VAR_INPUT
	ParamTempoTimeout				: TIME := T#20S;		(* (s) Tempo before timeout. *)
	IN_Directory 					: T_maxstring := 'C:\TwinCAT\Functions\Annex_Fonctions\SendEmail\';	// Directory of the SMTP.Exe file. 
	IN_Reset_OPC					: BOOL;					// Reset Mail server and alarms. 
	IN_Restart_Service_OPC			: BOOL;					// Restart SMTP services. 
	IN_ChangePhoneMailInfos_OPC		: BOOL;					// Change users Info (mails, name, Lvl, ... ) 
	FIFO							: FB_DBDatasetFifo;		// Buffer of the alarmes). 
	
END_VAR

VAR_OUTPUT
	OUT_Completed					: BOOL;		// Juste un trig pour dire que c'est fini. Written by the SMTP.Exe
	OUT_Error						: BOOL;		// Tant qu'il y a une erreur. Written by the SMTP.exe
	OUT_Busy						: BOOL;		// Envoi en cours. 
	OUT_NbMailSent 					: UINT;	// Number of mail being sent. 
END_VAR

VAR PERSISTENT
	AX_MailAddr						: ARRAY[1..CstNbUser] OF STRING(255);	//Contient tous les numéros des utilisateurs
	AX_Subscribed					: ARRAY[1..CstNbUser] OF BOOL		;	// List of subscription. 
	AX_NomUtili						: ARRAY[1..CstNbUser] OF STRING(50)	;	// List of user names. 
	AX_User_LVL						: ARRAY[1..CstNbUser] OF WORD;			//Contient tous les niveau d'adhésion des utilisateurs.
END_VAR

VAR_INPUT PERSISTENT
	ParamTempoRetry					: TIME := T#1M;  (* (s) Tempo before send email retry *) 
	ParamNetID						: STRING :='' ; (* AMS Net ID where the SMTP.exe file is stored *)
END_VAR

VAR

	// M_AlarmManager 
	MesDataExd.MesData			: ServerMail;
	RS_AlarmDestinator		: RS;
	
	// M_Write Param	
	bAlarmNoDestinator		: BOOL;
	bSendMail				: BOOL;
	
	bWriteParam				: BOOL;
	Body					: T_MaxString;
	MailAddr				: T_MaxString;
	MesTimeStamp			: STRING(17);	
	CalTimeStamp			: STRING(255);

	//M_Send
	SendMail				: NT_StartProcess;
	
	//M_OPC
	Trig_OPC				: R_TRIG;
	RS_OPC					: RS;
	Trig_Reset				: R_TRIG;

	KK						: UINT;
	NbDest					: INT;
	TON_Retry				: TON;
	Old_Count				: UDINT;
	R_TRIG_Retry			: R_TRIG;
	
END_VAR

M_AlarmManager();
M_OPC();
M_Evaluate();

IF IN_Reset_OPC THEN
	M_Reset();
END_IF
TON_Retry(IN := Old_Count = fifo.nCount AND NOT R_TRIG_Retry.Q, pt := ParamTempoRetry);

R_TRIG_Retry(clk := TON_Retry.Q);
IF old_count <> fifo.nCount THEN
	Old_Count := fifo.nCount;
END_IF
bWriteParam := fifo.nCount > 0; 	// if the buffer is not empty, send mail. 
fifo.A_Get();	// Get the next alarm to send. 

MesTimeStamp := CONCAT(REPLACE(STR1:= left(str := FIFO.Out.TimeStamp_Act, 16), STR2 := ' ', L := 1, P := 11), ' ') ;
ReplaceAll( In_StringTosearch := MesTimeStamp, In_StringToFind := '/', IN_StringToReplace := '-', OUT_StringToSearch => CalTimeStamp);

Body := concat(left(FIFO.Out.Message, 125),SEL(FIFO.Out.Value, ' : Desactive"',' : Active"')) ; 
Body := concat( STR1:= UINT_TO_STRING(FIFO.Out.ID) , STR2:= concat(STR1:=' ,' , STR2:=Body )) ; 
Body := concat( STR1:= 'ID:' , STR2:=Body ) ; 
Body := concat('"', Concat(CalTimeStamp,Body));


MailAddr := '"';
NbDest := 0;
FOR KK := 1 TO CstNbUser DO
	IF AX_Subscribed[KK] AND AX_MailAddr[KK] <> '' AND (AX_User_LVL[KK] AND Fifo.out.Alarms_LVL)>0 THEN		// If user is subscribed to this alarm, add his mail adress to the list. 
		IF MailAddr = '"' THEN
			MailAddr := concat('"', AX_MailAddr[KK]);	// Initialize first sender. 
		END_IF
		NbDest := NbDest + 1;
	END_IF
END_FOR

IF NbDest >0 THEN
	IF NbDest>1 THEN
		FOR KK := 1 TO CstNbUser DO
			IF AX_Subscribed[KK] AND MailAddr <> AX_MailAddr[KK] AND (AX_User_LVL[KK] AND Fifo.out.Alarms_LVL)>0 THEN
				MailAddr := concat(concat(MailAddr, ', '), AX_MailAddr[KK]);		// append other mail adress if several users subsribed to this alarm. 
			END_IF
		END_FOR
	END_IF
	MailAddr := concat(MailAddr, '" ');
	bSendMail := TRUE;
	bAlarmNoDestinator	:= FALSE;
ELSE 
	bAlarmNoDestinator	:= TRUE;
	bSendMail 			:= FALSE;

END_IF	

SendMail
(
	NETID := ParamNetID,
	PATHSTR := concat(IN_Directory, 'SMTP.exe'),
	DIRNAME := IN_Directory,
	COMNDLINE := concat(str1 := MailAddr, str2 := body),
	start := bSendMail AND bWriteParam and not TON_Retry.Q
);

IF OUT_Completed THEN 
	SendMail(start := FALSE);
	OUT_Completed := FALSE;
	OUT_NbMailSent := OUT_NbMailSent + 1;

	bSendMail := FALSE;
	FIFO.A_Remove();
END_IF	

IF OUT_NbMailSent > 30000 THEN
	OUT_NbMailSent := 0;
END_IF

METHOD M_AlarmManager
VAR
	
	FB_AlarmCodeManager : FB_AlarmCodeManager;

END_VAR
// Gestion des alarmes internes au code

RS_AlarmDestinator(SET:= bAlarmNoDestinator , RESET1:= IN_Reset_OPC ) ; 

FB_AlarmCodeManager
(
	bAlarm1 := RS_AlarmDestinator.Q1,			// No recipient for at least one alarm
	bAlarm2 := OUT_Error,						// Out Error to send mail
	bAlarm3 := SendMail.ERR,					// Execution of SenMail.exe did not work. 
	bAlarm4 := FIFO.bOverwrite,					// Fifo Overflow
	bAlarm5 :=FALSE,							//
	bAlarm6 :=FALSE,    						//
	bAlarm7 :=FALSE,    						//
	bAlarm8 :=FALSE,    						//
	bAlarm9 :=FALSE,    						//
	bAlarm10 :=FALSE,   						//
	bAlarm11 :=FALSE,   						//
	bAlarm12 :=FALSE,   						//
	bAlarm13 :=FALSE,   						//
	bAlarm14 :=FALSE,   						//
	bAlarm15 :=FALSE,							//	
	wAlarmCode =>MesData.MesAlarmCode
);
END_METHOD

METHOD M_Evaluate
VAR 
END_VAR

Mesdata.AX_MailAddr		:= AX_MailAddr			;
Mesdata.AX_Subscribed	:= AX_Subscribed	    ;
MesData.AX_NomUtili		:= AX_NomUtili		    ;
MesData.OUT_NbMailSent	:= OUT_NbMailSent		;
MesData.AX_UserLVL		:= AX_User_LVL		    ;
END_METHOD

METHOD M_Init : BOOL
VAR_INPUT
END_VAR
END_METHOD

METHOD M_OPC : BOOL
VAR

END_VAR
Trig_OPC(CLK := IN_ChangePhoneMailInfos_OPC);
RS_OPC(SET:= Trig_OPC.Q);

//TrigRestartService(CLK := IN_Restart_Service_OPC);
//FUN_RestartStunnel(IN_Start := TrigRestartService.Q, IN_Directory := IN_Directory);


IF RS_OPC.Q1 THEN
	// Numéro de téléphone
	AX_MailAddr := OpcUa.AllValueW.AX_MailAddr_OPC;
	
	// Nom d'utilisateur
	AX_NomUtili	:= OpcUa.AllValueW.AX_NamesUsers_OPC;
	
	// User LVL . 
	AX_User_LVL := OpcUa.AllValueW.AX_UserLVL;
	
	// Mise a jour de la liste des subscribed
	AX_Subscribed := OpcUa.AllValueW.AX_SubscribedMail_OPC;

	RS_OPC(RESET1:= TRUE);
	RS_OPC(Reset1 := FALSE);
END_IF

Trig_Reset(CLK := IN_Reset_OPC);
IN_Reset_OPC := Trig_Reset.Q;
END_METHOD

METHOD M_Reset : BOOL
VAR_INPUT
END_VAR
VAR
	

END_VAR
FIFO.A_Reset();
IN_Reset_OPC 			:= FALSE;
bAlarmNoDestinator 		:= FALSE ;	
bSendMail				:= FALSE;
SendMail(Start:= FALSE ) ;
END_METHOD

END_PROGRAM

// ---- 00_FunctionsBlocks/Communication/ModbusRTU/CheckStruct.TcPOU
FUNCTION CheckStruct : BOOL
//Allows to compare 2 Struct_InputRTU, TRUE if struct are the same
VAR_INPUT
	InStruct1 : Struct_InputRTU;
	InStruct2 : Struct_InputRTU;
END_VAR
VAR
	bCompareBuffer 	: BOOL := TRUE;
	KK 				: UINT;
	AdrNull			: Pointer to array[1..125] of word;
END_VAR

IF InStruct1.InBuffer <> adrNull AND instruct2.InBuffer <> AdrNull THEN
	CheckStruct:= MEMCMP(pBuf1 := ADR(instruct1), pBuf2 := ADR(InStruct2), n := SIZEOF(InStruct1)) = 0;

	//FOR KK := 1 TO 125 DO
	//	bCompareBuffer := bCompareBuffer AND (InStruct1.InBuffer^[KK] = InStruct2.InBuffer^[KK]);
	//END_FOR
	//
	//
	//CheckStruct :=(InStruct1.InStartAddr	= InStruct2.InStartAddr	AND InStruct1.InQuantity	= InStruct2.InQuantity	AND InStruct1.InUnitID	    = InStruct2.InUnitID	AND  bCompareBuffer AND InStruct1.InFunction	= InStruct2.InFunction	);
END_IF

END_FUNCTION

// ---- 00_FunctionsBlocks/Communication/ModbusRTU/FB_ModbusRTU.TcPOU
FUNCTION_BLOCK FB_ModbusRTU
// Send Modbus Read Request for the first element of the buffer . Then remove the first line when executed ( busy)  and move all the other line to the left. Position 2 becomes position 1 , ...
VAR CONSTANT
	NbElementsBuffer				: UINT := 20;
	
END_VAR

VAR
	Buffer 							: ARRAY[1..NbElementsBuffer] OF Struct_InputRTU ; // Buffer to store actions
	Priority 						: ARRAY[1..NbElementsBuffer] OF UINT; // Array to store priorities
	InitialStruct 					: Struct_InputRTU;
	bInit 							: BOOL;
	ReadRTU1						: FB_ReadModbusRTU_V2;

	KK : UINT;
	
	pBoolNull						: BOOL;
	pIntNull						: INT;
	pArrayNull						: BYTE;

	R_TRIG_Error					: R_TRIG ;
	
END_VAR

IF NOT bInit THEN
	// Empty all structures . 
	M_Init();
ELSE
	
		// ATTENTION , IL NE FAUT PAS ENVOYER UN NOUVEAU MODBUS TANT QUE LE PRECEDENT N EST PAS FINI DE TRAITER .DE MEME IL NE FAUT PAS QUE LE CYCLE D AJOUT DU FIFO SOIT PLUS RAPIDE QUE LE TRAITEMENT DU RTU 
		// TEmpo de 30 s apres une alarmes avant de refaire un essai . il ne faudrait pas que ca bloque les autres commandes .  

		IF priority[1] <> 0 THEN

			ReadRTU1(
				InClockRead := TRUE,
				InStartAddr := Buffer[1].InStartAddr,
				InQuantity := Buffer[1].InQuantity,
				InUnitID := Buffer[1].InUnitID,
				InTimeout := T#500MS,
				InAddrDest := Buffer[1].InBuffer,
				InFunctionRead := Buffer[1].InFunction
			);
		END_IF
		
		
		
		MEMCPY(destAddr := Buffer[1].OutBusy, srcAddr := ADR(ReadRTU1.OutBusy), n := SIZEOF(ReadRTU1.OutBusy));		

		//R_TRIG_Error(CLK:= ReadRTU1.OutErrorMbRead) ; 
		
		IF ReadRTU1.OutbCompleted OR ReadRTU1.OutErrorMbRead THEN	// La lecture s 'est terminée par une erreur ou correcteemnt, on passe à l'element du buffer suivant . 
			MEMCPY(destAddr := Buffer[1].OutError, srcAddr := ADR(ReadRTU1.OutErrorMbRead), n := SIZEOF(ReadRTU1.OutErrorMbRead)); // Copy the errOR  
			MEMCPY(destAddr := Buffer[1].OutErrorId, srcAddr := ADR(ReadRTU1.OutErrorId), n := SIZEOF(ReadRTU1.OutErrorId));
			MEMCPY(destAddr := Buffer[1].OutCompleted, srcAddr := ADR(ReadRTU1.OutbCompleted), n := SIZEOF(ReadRTU1.OutbCompleted));	
			ReadRTU1.InClockRead := FALSE ; 
			ReadRTU1.Reset		:= TRUE ; 
			M_DeleteAction(InLigne := 1);
			//R_TRIG_Error(CLK:= FALSE ) ; 
			
		END_IF
END_IF

METHOD M_AddAction_FIFO : UINT //Method to add an element with a priority using FIFO strategy

VAR_INPUT
	InStruct 		: Struct_InputRTU;		// Structure input
	InPriority 		: UINT;					// Strategy input
END_VAR
VAR_OUTPUT
	OutBusy 		: BOOL;					// Output state of the Method
	OutError 		: BOOL;					// Output error of the Method
	OutErrorID 		: UINT;					//1: Empty input 2: Full Buffer
	OutCompleted 	: BOOL;					// Output state of the Method : not busy and no error
END_VAR
VAR
	KK 				: UINT;
	LineToDelete	: UINT;
END_VAR
OutError 	:= FALSE;
OutBusy 	:= TRUE;

IF NOT (CheckStruct(InStruct1 := InitialStruct, InStruct2 := InStruct)) AND InPriority <> 0 THEN 			// Check that we don't input an empty value
	IF CheckStruct(InStruct1 := buffer[NbElementsBuffer], InStruct2 := InitialStruct) THEN 			// Check that the buffer isn't already full
		FOR KK := 1 TO NbElementsBuffer - 1 DO
			IF NOT CheckStruct(InStruct1 := buffer[NbElementsBuffer-KK], InStruct2 := InitialStruct) AND Priority[NbElementsBuffer-KK] > InPriority THEN 			// If the next position isn't empty  
				buffer[NbElementsBuffer-KK+1] := buffer[NbElementsBuffer-KK]; 		// I replace this position by the next  ( CE PREMIER IF N EST PAS EXECUTER SI TOUTES LES PRIORITES SONT IDENTIQUES . )
				Priority[NbElementsBuffer -KK +1 ] := Priority[NbElementsBuffer-KK];
			ELSE
				IF NOT CheckStruct(InStruct1 := buffer[NbElementsBuffer-KK], InStruct2 := InitialStruct) THEN		// Detect for buffer element that is not empty and assign new element to read to it. 
					buffer[NbElementsBuffer-KK+1] 	:= InStruct;
					M_AddAction_FIFO 				:= NbElementsBuffer-KK+1;
					Priority[NbElementsBuffer-KK+1] := InPriority;
					OutCompleted 		:= TRUE;
					EXIT ;
				END_IF
			END_IF
		END_FOR
		IF NOT Outcompleted THEN
			buffer[1] := InStruct;
			Priority[1] := InPriority;
			OutCompleted := TRUE;
			M_AddAction_Fifo := 1;
		END_IF
	ELSE
		OutErrorID 	:= 2;
		OutError 	:= TRUE;
	END_IF
ELSE
	OutErrorID 	:= 1;
	OutError 	:= TRUE;
END_IF
IF M_VerifActions(OutLigne=>LineToDelete) THEN	// Verifie si il  n ya pas deux fois la meme ligne , sinon, supprime les lignes en doubles . En pratique, forcement la derniere ligne . 
	M_DeleteAction(InLigne := LineToDelete);
END_IF
OutBusy := FALSE;
END_METHOD

METHOD M_DeleteAction : BOOL
VAR_INPUT
	InLigne 	: UINT;			// Input Ligne to delete
END_VAR
VAR_OUTPUT
	OutBusy 		: BOOL;					// Output state of the Method
	OutError 		: BOOL;					// Output error of the Method
	OutErrorID 		: UINT;					// 1: InLigne greater than Buffer size, 2: The buffer ligne is already empty, 3: The buffer is full
	OutCompleted 	: BOOL;					// Output state of the Method : not busy and no error
	
END_VAR

VAR
	KK 				: UINT;
END_VAR
IF InLigne <= NbElementsBuffer THEN // Check the InLigne is in the range of the buffer
	IF NOT checkstruct(InStruct1 := buffer[InLigne], InStruct2 := InitialStruct) THEN	// Check that the buffer ligne is not already empty
		IF checkstruct(InStruct1 := buffer[NbElementsBuffer], InStruct2 := InitialStruct)THEN //check that the buffer is not full
			FOR KK := InLigne TO NbElementsBuffer -1 DO
				Buffer[KK] := buffer[KK + 1] ;
				Priority[KK] := Priority[KK + 1] ;
			END_FOR
		ELSE
			OutError := TRUE;
			OutBusy := FALSE;
			OutCompleted := FALSE;
			OutErrorID := 3;
		END_IF
	ELSE
		OutError := TRUE;
		OutCompleted := FALSE;
		OutBusy := TRUE;
		OutErrorID := 2;
		
	END_IF
ELSE
	OutCompleted := FALSE;
	OutError := TRUE;
	OutBusy := FALSE;
	OutErrorID := 1;
END_IF
END_METHOD

METHOD M_Init : BOOL
VAR
	InStruct : Struct_InputRTU;
END_VAR

// Initialize the structure with empty elements. 

InitialStruct.InBuffer := ADR(pArrayNull);
InitialStruct.OutBusy := ADR(pBoolNull);
InitialStruct.OutCompleted := ADR(pBoolNull);
InitialStruct.OutError := ADR(pBoolNull);
InitialStruct.OutErrorId := ADR(pIntNull);
FOR KK := 1 TO NbElementsBuffer DO 
	Buffer[KK] := InitialStruct;
END_FOR	

bInit := TRUE;
END_METHOD

METHOD M_VerifActions : BOOL // Verifies there is not repeat in the liste : TRUE = At least 2 elements are the same
VAR_OUTPUT
	OutLigne 	 : UINT;
END_VAR

VAR
	KK: UINT;
	JJ: UINT;
	CheckStructValue : BOOL;
END_VAR
FOR KK := 1 TO NbElementsBuffer DO
	FOR JJ := 1 + KK TO NbElementsBuffer DO
		IF CheckStruct(InStruct1 := InitialStruct, instruct2 := buffer[KK]) THEN
			EXIT;
		ELSE
			CheckStructValue :=  checkstruct(InStruct1 := buffer[JJ], InStruct2 := buffer[KK]);
			M_VerifActions := M_VerifActions OR (CheckStructValue ) ;
			OutLigne := SEL(CheckStructValue AND Priority[KK]> priority[JJ], KK, JJ);
		END_IF
	END_FOR
END_FOR
END_METHOD

END_FUNCTION_BLOCK

// ---- 00_FunctionsBlocks/Communication/ModbusRTU/FB_ReadModbusRTU_V2.TcPOU
FUNCTION_BLOCK FB_ReadModbusRTU_V2
/////////////////////////////////////////////////////////////////////// 
///////Read Modbus RTU on Rising Edge of Trigger ClockRead ////////
//If there is lost of communication, ParamNbAlms then if still 
//error wait ParamTimeRetry then loop 
//Version : V1.1
///////////////////////////////////////////////////////////////////////

VAR_INPUT
	InClockRead 			: BOOL;  		// Boolean to start the read
	InStartAddr				: WORD;  		// First address of the block
	InQuantity			    : WORD;	 		// Quantity of registers to read
	InUnitID				: BYTE ; 		// Unit Id of the Slave to be read
	InTimeout 				: TIME:=T#2S;   // Timeout param for the read
	InAddrDest		        : POINTER TO BYTE;
	InFunctionRead          : UINT;          // 0 := ReadInputRegs, 1 := ReadRegs 
	ParamEnableRetryPause	: BOOL ; 
	Reset					: BOOL ;
END_VAR

VAR_OUTPUT
	OutErrorMbRead  		: BOOL; 	                // Alarm if three modbus attempts failed.
	OutBusy					: BOOL;					    //Busy
	OutErrorId				: INT;            //Id number of the error based on TC
	OutbCompleted			: BOOL;
	TmpError				: BOOL;	
END_VAR

VAR
	//Parameters
	ParamNbAlms				: UINT := 3;				// Parameter for the number of retries before the alarme
	ParamTimeRetry 			: TIME:=T#30S;				//Time to wait before a retry
	
	//Instantiation of FB
	MB 						: ModbusRtuMaster_PcCOM; 		// Multiple registers reading FROM SUB9 Interface
	MB_EL					: ModbusRtuMasterV2_KL6x22B;  // Multiple registers reading FROM EL6021 Interface
	R_TRIG          		: R_TRIG; 					// Rising edge detection for the trigger.
	TempoRetry      		: TP;
	
	//Variables of the code 
	Step            		: INT; 		    			// Grafcet step
	AlarmCounter    		: UINT; 					// Alarm Counter. Incremennted if modbus errOR  Alarm if counter =3 , resetable.  
	bRetry          		: BOOL:= FALSE; 			// Boolean to denote the retries
	
	TmpBusy					: BOOL;
	TmpErrorId				: INT;	
	
	TON_ReadRTU						: TON; 
END_VAR

OutbCompleted:= FALSE;
// RESET //
	IF Reset THEN 
			AlarmCounter		:= MAX(0,AlarmCounter-1) ;	// on enleve 1 au compteur pour supprimer l'alamrme. 
			OutErrorId 			:= 0 ; 
			OutErrorMbRead 	:=FALSE;
			Reset 				:= FALSE;
	END_IF
	
// ALARM MANAGEMENT //
TempoRetry(PT := ParamTimeRetry);
IF AlarmCounter = ParamNbAlms THEN 
	OutErrorMbRead 	:=TRUE;
	bRetry := SEL(ParamEnableRetryPause , FALSE ,  TRUE);		// False = disable retry 	
ELSE
	bRetry := FALSE;
	
END_IF

	// MODBUS SEQUENCE //
	CASE step OF
		0://Idle
			R_TRIG(CLK := InClockRead);
			IF R_TRIG.Q THEN 
				R_TRIG(CLK := FALSE);
				Step :=1;
				OutBusy         := TRUE;
			END_IF
		1 ://Processing Reply  
			TON_ReadRTU(IN:= TRUE , PT:= InTimeout + T#100MS ) ; // Overlay timeout . 
	    	CASE InFunctionRead OF
				1: 
					MB_EL.ReadCoils
					(
						UnitID := InUnitId, 
						Quantity := InQuantity, 
						MBAddr := InStartAddr, 
						cbLength := 2* InQuantity, 
						pMemoryAddr := InAddrDest, 
						Execute := TRUE, 
						Timeout := InTimeout,
						Error => TmpError,
						Busy => TmpBusy,
						ErrorId => TmpErrorId,
					);	
				2:
					MB_EL.ReadInputStatus
					(
						UnitID := InUnitId, 
						Quantity := InQuantity, 
						MBAddr := InStartAddr, 
						cbLength := 2* InQuantity, 
						pMemoryAddr := InAddrDest, 
						Execute := TRUE, 
						Timeout := InTimeout,
						Error => TmpError,
						Busy => TmpBusy,
						ErrorId => TmpErrorId,
					);	
				3:
					MB_EL.ReadRegs
					(
						UnitID := InUnitId, 
						Quantity := InQuantity, 
						MBAddr := InStartAddr, 
						cbLength := 2* InQuantity, 
						pMemoryAddr := InAddrDest, 
						Execute := TRUE, 
						Timeout := InTimeout,
						Error => TmpError,
						Busy => TmpBusy,
						ErrorId => TmpErrorId,
					  );
				4:
					MB_EL.ReadInputRegs
					(
						UnitID := InUnitId, 
						Quantity := InQuantity, 
						MBAddr := InStartAddr, 
						cbLength := 2* InQuantity, 
						pMemoryAddr := InAddrDest, 
						Execute := TRUE, 
						Timeout := InTimeout,
						Error => TmpError,
						Busy => TmpBusy,
						ErrorId => TmpErrorId,
					);
				5:
					MB_EL.WriteSingleCoil
					(
						UnitID := InUnitId, 
						Quantity := InQuantity, 
						MBAddr := InStartAddr, 
						cbLength := 2* InQuantity, 
						pMemoryAddr := InAddrDest, 
						Execute := TRUE, 
						Timeout := InTimeout,
						Error => TmpError,
						Busy => TmpBusy,
						ErrorId => TmpErrorId,
					);
				6:
					MB_EL.WriteSingleRegister
					(
						UnitID := InUnitId, 
						Quantity := InQuantity, 
						MBAddr := InStartAddr, 
						cbLength := 2* InQuantity, 
						pMemoryAddr := InAddrDest, 
						Execute := TRUE, 
						Timeout := InTimeout,
						Error => TmpError,
						Busy => TmpBusy,
						ErrorId => TmpErrorId,
					);
				15:
					MB_EL.WriteMultipleCoils
					(
						UnitID := InUnitId, 
						Quantity := InQuantity, 
						MBAddr := InStartAddr, 
						cbLength := 2* InQuantity, 
						pMemoryAddr := InAddrDest, 
						Execute := TRUE, 
						Timeout := InTimeout,
						Error => TmpError,
						Busy => TmpBusy,
						ErrorId => TmpErrorId,
					);
				16:
					MB_EL.WriteRegs
					(
						UnitID := InUnitId, 
						Quantity := InQuantity, 
						MBAddr := InStartAddr, 
						cbLength := 2* InQuantity, 
						pMemoryAddr := InAddrDest, 
						Execute := TRUE, 
						Timeout := InTimeout,
						Error => TmpError,
						Busy => TmpBusy,
						ErrorId => TmpErrorId,
					);
			END_CASE
			
			IF NOT (TmpBusy) AND NOT (TmpError) THEN
				TempoRetry(In:= FALSE);
				TON_ReadRTU(IN:= FALSE ) ; 
				MB_EL.ReadInputRegs(Execute:= FALSE);
				MB_EL.ReadRegs(Execute:= FALSE);
				MB_EL.ReadCoils(Execute:= FALSE);
				MB_EL.ReadInputStatus(Execute:= FALSE);
				MB_EL.WriteSingleCoil(Execute:= FALSE);
				MB_EL.WriteSingleRegister(Execute:= FALSE);
				MB_EL.WriteMultipleCoils(Execute:= FALSE);
				MB_EL.WriteRegs(Execute:= FALSE);
				OutErrorId 		:= 0;
				OutErrorMbRead	:= FALSE;
				AlarmCounter	:= 0; // Reset counter after successful modbus read. 
				OutbCompleted 	:= TRUE ; 
				Step 			:= 0;
				OutBusy         := FALSE;
			ELSIF ((NOT (TmpBusy) AND TmpError) OR TON_ReadRTU.Q)  AND NOT(bRetry) THEN

				TempoRetry(In:= FALSE);
				bRetry := FALSE;
				MB_EL.ReadCoils(Execute:= FALSE);
				MB_EL.ReadInputRegs(Execute:= FALSE);
				MB_EL.ReadInputStatus(Execute:= FALSE);
				MB_EL.ReadRegs(Execute:= FALSE);
				MB_EL.WriteSingleCoil(Execute:= FALSE);
				MB_EL.WriteSingleRegister(Execute:= FALSE);
				MB_EL.WriteMultipleCoils(Execute:= FALSE);
				MB_EL.WriteRegs(Execute:= FALSE);
				AlarmCounter 	:= MIN(AlarmCounter + 1,3) ; 
				OutErrorId		:= SEL(TON_ReadRTU.Q , TmpErrorId ,250 );
				Step 			:= 0;
				TON_ReadRTU(IN:= FALSE ) ; 
				OutBusy         := FALSE;
			ELSIF NOT (TmpBusy) AND TmpError AND bRetry THEN
				MB_EL.ReadInputRegs(Execute:= FALSE);
				MB_EL.ReadRegs(Execute:= FALSE);
				MB_EL.ReadCoils(Execute:= FALSE);
				MB_EL.ReadInputStatus(Execute:= FALSE);
				MB_EL.WriteSingleCoil(Execute:= FALSE);
				MB_EL.WriteSingleRegister(Execute:= FALSE);
				MB_EL.WriteMultipleCoils(Execute:= FALSE);
				MB_EL.WriteRegs(Execute:= FALSE);
				step := 2;
				OutBusy         := FALSE;
			END_IF	
		2: 
			TempoRetry(In:= TRUE);		// LEAVE SOME TIME BEFORE NEW ATTEMPT . 
			IF NOT(TempoRetry.Q) THEN
				TempoRetry(In:= FALSE);
				//AlarmCounter := 0;
				step := 0;
				
			END_IF
			
	END_CASE

END_FUNCTION_BLOCK

// ---- 00_FunctionsBlocks/Communication/ModbusRTU/Sample_ModbusRTU.TcPOU
PROGRAM Sample_ModbusRTU
VAR
	ModbusRTU				: FB_ModbusRTU;
	MesBlock				: ARRAY[1..8] OF ARRAY[1..120] OF WORD;	
	AX_Addr					: ARRAY[1..8] OF UINT 	:= [1,		1,		1,		1,		1, 		1, 		1, 		1];
	AX_Qty					: ARRAY[1..8] OF UINT	:= [1,		1,		1,		1,		1, 		1, 		1, 		1];
	AX_UnitId				: ARRAY[1..8] OF BYTE	:= [1,		1,		1,		1,		1, 		1, 		1, 		1];
	AX_Function				: ARRAY[1..8] OF UINT	:= [1,		2,		3,		4,		5, 	 	6, 	 	15, 	16];	
	AX_Priority				: ARRAY[1..8] OF UINT	:= [1,		1,		1,		1,		1, 	 	1, 	 	1, 		1 ];
	AX_bStart				: ARRAY[1..8] OF BOOL;
	MbStruct				: ARRAY[1..8] OF Struct_InputRTU;	
	
	KK: INT;
END_VAR

ModbusRTU();

FOR KK := 1 TO 8 DO 
	MbStruct[KK].InBuffer := ADR(MesBlock[KK]);
	MbStruct[KK].InFunction := AX_Function[KK];
	MbStruct[KK].InQuantity := AX_Qty[KK];
	MbStruct[KK].InStartAddr := AX_Addr[KK];
	MbStruct[KK].InUnitID := AX_UnitId[KK];
END_FOR


IF CalLocalTimeStruct.wSecond MOD 5 = 0 THEN
	FOR KK := 1 TO 8 DO
		IF AX_bStart[KK] THEN
			ModbusRTU.M_AddAction_FIFO(InStruct := MbStruct[KK], InPriority := AX_Priority[KK]);
		END_IF
	END_FOR
	
END_IF

END_PROGRAM

// ---- 00_FunctionsBlocks/Communication/ModbusTCP/FB_ModbusRead.TcPOU
FUNCTION_BLOCK FB_ModbusRead
////////////////// 
// Read Modbus TCP/IP on Rising Edge of Trigger ClockRead. Returns alarm and stop modbus Read after three consecutive Modbus attempts that failed. 
//////////////////

VAR_INPUT
	
	// Modbus ReadRegs FB inputs
	pDestAddr 	: POINTER TO BYTE ; // Pointer to variable in which the read data have to be stored
	sIPAddr 	: STRING(15);		// Modbus server device IP adress
	tTimeout 	: TIME;				// Timeout
	nTcpPort 	: UINT;
	nQuantity 	: WORD;				// Quantity of words to be read
	nMBAddr 	: WORD ;			// Starting Register adress
	
	cbLength 	: UDINT;			// Length of variable to host the read data
	nUnitID 	: BYTE;				// Unit ID in case of serial connexion after modbus server. Usually equals to 1
	
	ClockRead	: BOOL; 			// Rising Edge Modbus Trigger
	Reset		: BOOL; 			// Reset Trigger to clean alarm and counter.
	
	ParamTimeRetry 			: TIME:=T#30S;				//Time to wait before a retry
	ParamNbAlms				: INT := 3;				// Parameter for the number of retries before the alarme
	ParamEnableRetryPause	: BOOL ; 
	
	
END_VAR

VAR_OUTPUT
	ErrorId			: UDINT;	// Error Id returned by FB ( see ADS error Code ) . 
	
	Busy			: BOOL ;	// FB busy to proceed command
	ModbusReadAlarm	: BOOL; 	// Alarm if three modbus attempt failed.
	OUT_NbRead		: UDINT;
END_VAR

VAR
	R_TRIG 				: R_TRIG; 			// Rising edge detection for the trigger.
	FB_MBReadRegs 		: FB_MBReadRegs; 	// Multiple registers reading
	
	Step				: INT; 				// Grafcet step
	AlarmCounter		: INT; 				// Alarm Counter. Incremennted if modbus errOR  Alarm if counter =3 , resetable.  

	TempoRetry      		: TP;

	bRetry          		: BOOL:= FALSE; 			// Boolean to denote the retries	
END_VAR

// ALARM MANAGEMENT //
TempoRetry(PT := ParamTimeRetry);
	IF AlarmCounter=ParamNbAlms THEN 
		ModbusReadAlarm 	:=TRUE;
		bRetry := SEL(ParamEnableRetryPause , FALSE ,  TRUE);		// False = disable retry 		
	ELSE
		ModbusReadAlarm := FALSE;
		ErrorId			:= 0;
		bRetry := FALSE;		// False = disable retry 	
	END_IF


// MODBUS SEQUENCE //
CASE Step OF 
	0:
		R_TRIG(CLK :=ClockRead);
		
		IF R_TRIG.Q THEN 
			Step :=1;
			Busy := TRUE;
			OUT_NbRead := 0;
		END_IF
	1:
	   FB_MBReadRegs(
	  			sIPAddr:= sIPAddr , 
				nTCPPort:= nTcpPort ,
				nUnitID:= nUnitID,
				nQuantity:= nQuantity,
				nMBAddr:= nMBAddr, 
				cbLength:= cbLength, 
				pDestAddr:= pDestAddr, 
				bExecute:= TRUE,
				tTimeout:= tTimeout,
				cbRead => OUT_NbRead
				);
				
		IF NOT FB_MBReadRegs.bBusy AND NOT FB_MBReadRegs.bError THEN
			FB_MBReadRegs(bExecute:= FALSE);
			AlarmCounter	:=0; // Reset counter after successful modbus read. 
			Step 			:=0;
			Busy := FALSE;
		ELSIF NOT FB_MBReadRegs.bBusy AND FB_MBReadRegs.bError AND NOT(bRetry) THEN
			FB_MBReadRegs(bExecute:= FALSE);
			AlarmCounter 	:= MIN(AlarmCounter+1,ParamNbAlms) ; 
			ErrorId			 :=FB_MBReadRegs.nErrId;
			Step 			:=0;
			Busy := FALSE;
			TempoRetry(In:= FALSE);
			bRetry := FALSE;
		ELSIF NOT FB_MBReadRegs.bBusy AND FB_MBReadRegs.bError AND bRetry THEN
			FB_MBReadRegs(bExecute:= FALSE);
			step := 2;
			Busy := FALSE;		
		END_IF	
	2: 
		TempoRetry(In:= TRUE);		// LEAVE SOME TIME BEFORE NEW ATTEMPT . 
		IF NOT(TempoRetry.Q) THEN
			TempoRetry(In:= FALSE);
			//AlarmCounter := 0;
			step := 0;
			
		END_IF
		
END_CASE

// RESET //
	IF Reset THEN 
			AlarmCounter 		:= 0 ; 
			ErrorId 			:= 0 ; 
			ModbusReadAlarm 	:=FALSE;
			Reset 				:= FALSE;
	END_IF

// BUSY //

END_FUNCTION_BLOCK

// ---- 00_FunctionsBlocks/Communication/ModbusTCP/FB_ModbusReadCoils.TcPOU
FUNCTION_BLOCK FB_ModbusReadCoils
////////////////// 
// Read Modbus TCP/IP on Rising Edge of Trigger ClockRead. Returns alarm and stop modbus Read after three consecutive Modbus attempts that failed. 
//////////////////

VAR_INPUT
	
	// Modbus ReadRegs FB inputs
	pDestAddr 	: POINTER TO BYTE ; // Pointer to variable in which the read data have to be stored
	sIPAddr 	: STRING(15);		// Modbus server device IP adress
	tTimeout 	: TIME;				// Timeout
	nTcpPort 	: UINT;
	nQuantity 	: WORD;				// Quantity of words to be read
	nMBAddr 	: WORD ;			// Starting Register adress
	
	cbLength 	: UDINT;			// Length of variable to host the read data
	nUnitID 	: BYTE;				// Unit ID in case of serial connexion after modbus server. Usually equals to 1
	
	ClockRead	: BOOL; 			// Rising Edge Modbus Trigger
	Reset		: BOOL; 			// Reset Trigger to clean alarm and counter.
	
END_VAR

VAR_OUTPUT
	ErrorId			: UDINT;	// Error Id returned by FB ( see ADS error Code ) . 
	
	Busy			: BOOL ;	// FB busy to proceed command
	ModbusReadAlarm	: BOOL; 	// Alarm if three modbus attempt failed.
	OUT_NbRead		: UDINT;
END_VAR

VAR
	R_TRIG 				: R_TRIG; 			// Rising edge detection for the trigger.
	FB_MBReadCoils 		: FB_MBReadCoils; 	// Multiple registers reading
	
	Step				: INT; 				// Grafcet step
	AlarmCounter		: INT; 				// Alarm Counter. Incremennted if modbus errOR  Alarm if counter =3 , resetable.  

	
END_VAR

// ALARM MANAGEMENT //

	IF AlarmCounter=3 THEN 
		ModbusReadAlarm 	:=TRUE;
		
	ELSE
		ModbusReadAlarm := FALSE;
		ErrorId			:= 0;
		
	END_IF


// MODBUS SEQUENCE //
CASE Step OF 
	0:
		R_TRIG(CLK :=ClockRead);
		
		IF R_TRIG.Q THEN 
			Step :=1;
			Busy := TRUE;
			OUT_NbRead := 0;
		END_IF
	1:
	   FB_MBReadCoils(
	  			sIPAddr:= sIPAddr , 
				nTCPPort:= nTcpPort ,
				nUnitID:= nUnitID,
				nQuantity:= nQuantity,
				nMBAddr:= nMBAddr, 
				cbLength:= cbLength, 
				pDestAddr:= pDestAddr, 
				bExecute:= TRUE,
				tTimeout:= tTimeout,
				cbRead => OUT_NbRead
				);
				
		IF NOT FB_MBReadCoils.bBusy AND NOT FB_MBReadCoils.bError THEN
			FB_MBReadCoils(bExecute:= FALSE);
			AlarmCounter	:=0; // Reset counter after successful modbus read. 
			Step 			:=0;
			Busy := FALSE;
		ELSIF NOT FB_MBReadCoils.bBusy AND FB_MBReadCoils.bError THEN
			FB_MBReadCoils(bExecute:= FALSE);
			AlarmCounter 	:= MIN(AlarmCounter+1,3) ; 
			ErrorId			 :=FB_MBReadCoils.nErrId;
			Step 			:=0;
			Busy := FALSE;
		END_IF
		
END_CASE

// RESET //
	IF Reset THEN 
			AlarmCounter 		:= 0 ; 
			ErrorId 			:= 0 ; 
			ModbusReadAlarm 	:=FALSE;
			Reset 				:= FALSE;
			FB_MBReadCoils		(bExecute := FALSE);
	END_IF

// BUSY //

END_FUNCTION_BLOCK

// ---- 00_FunctionsBlocks/Communication/ModbusTCP/FB_ModbusReadInput.TcPOU
FUNCTION_BLOCK FB_ModbusReadInput
////////////////// 
// Read Modbus TCP/IP on Rising Edge of Trigger ClockRead. Returns alarm and stop modbus Read after three consecutive Modbus attempts that failed. 
//////////////////

VAR_INPUT
	
	// Modbus ReadRegs FB inputs
	pDestAddr 	: POINTER TO BYTE ; // Pointer to variable in which the read data have to be stored
	sIPAddr 	: STRING(15);		// Modbus server device IP adress
	tTimeout 	: TIME;				// Timeout
	nTcpPort 	: UINT;
	nQuantity 	: WORD;				// Quantity of words to be read
	nMBAddr 	: WORD ;			// Starting Register adress
	
	cbLength 	: UDINT;			// Length of variable to host the read data
	nUnitID 	: BYTE;				// Unit ID in case of serial connexion after modbus server. Usually equals to 1
	
	ClockRead	: BOOL; 			// Rising Edge Modbus Trigger
	Reset		: BOOL; 			// Reset Trigger to clean alarm and counter.
	
END_VAR

VAR_OUTPUT
	ErrorId			: UDINT;	// Error Id returned by FB ( see ADS error Code ) . 
	
	Busy			: BOOL ;	// FB busy to proceed command
	ModbusReadAlarm	: BOOL; 	// Alarm if three modbus attempt failed.
	OUT_NbRead		: UDINT;
END_VAR

VAR
	R_TRIG 				: R_TRIG; 			// Rising edge detection for the trigger.
	FB_MBReadInputs 		: FB_MBReadInputs; 	// Multiple registers reading
	
	Step				: INT; 				// Grafcet step
	AlarmCounter		: INT; 				// Alarm Counter. Incremennted if modbus errOR  Alarm if counter =3 , resetable.  

	
END_VAR

// ALARM MANAGEMENT //

	IF AlarmCounter=3 THEN 
		ModbusReadAlarm 	:=TRUE;
		
	ELSE
		ModbusReadAlarm := FALSE;
		ErrorId			:= 0;
		
	END_IF


// MODBUS SEQUENCE //
CASE Step OF 
	0:
		R_TRIG(CLK :=ClockRead);
		
		IF R_TRIG.Q THEN 
			Step :=1;
			Busy := TRUE;
			OUT_NbRead := 0;
		END_IF
	1:
	   FB_MBReadInputs(
	  			sIPAddr:= sIPAddr , 
				nTCPPort:= nTcpPort ,
				nUnitID:= nUnitID,
				nQuantity:= nQuantity,
				nMBAddr:= nMBAddr, 
				cbLength:= cbLength, 
				pDestAddr:= pDestAddr, 
				bExecute:= TRUE,
				tTimeout:= tTimeout,
				cbRead => OUT_NbRead
				);
				
		IF NOT FB_MBReadInputs.bBusy AND NOT FB_MBReadInputs.bError THEN
			FB_MBReadInputs(bExecute:= FALSE);
			AlarmCounter	:=0; // Reset counter after successful modbus read. 
			Step 			:=0;
			Busy := FALSE;
		ELSIF NOT FB_MBReadInputs.bBusy AND FB_MBReadInputs.bError THEN
			FB_MBReadInputs(bExecute:= FALSE);
			AlarmCounter 	:= MIN(AlarmCounter+1,3) ; 
			ErrorId			 :=FB_MBReadInputs.nErrId;
			Step 			:=0;
			Busy := FALSE;
		END_IF
		
END_CASE

// RESET //
	IF Reset THEN 
			AlarmCounter 		:= 0 ; 
			ErrorId 			:= 0 ; 
			ModbusReadAlarm 	:=FALSE;
			Reset 				:= FALSE;
			FB_MBReadInputs		(bExecute := FALSE);
	END_IF

// BUSY //

END_FUNCTION_BLOCK

// ---- 00_FunctionsBlocks/Communication/ModbusTCP/FB_ModbusReadInputRegs.TcPOU
FUNCTION_BLOCK FB_ModbusReadInputRegs
////////////////// 
// Read Modbus TCP/IP on Rising Edge of Trigger ClockRead. Returns alarm and stop modbus Read after three consecutive Modbus attempts that failed. 
//////////////////

VAR_INPUT
	
	// Modbus ReadRegs FB inputs
	pDestAddr 	: POINTER TO BYTE ; // Pointer to variable in which the read data have to be stored
	sIPAddr 	: STRING(15);		// Modbus server device IP adress
	tTimeout 	: TIME;				// Timeout
	
	nTCPport	: UINT:= 502;		// TCP Port
	
	nQuantity 	: WORD;				// Quantity of words to be read
	nMBAddr 	: WORD ;			// Starting Register adress
	
	cbLength 	: UDINT;			// Length of variable to host the read data
	nUnitID 	: BYTE;				// Unit ID in case of serial connexion after modbus server. Usually equals to 1
	
	ClockRead	: BOOL; 			// Rising Edge Modbus Trigger
	Reset		: BOOL; 			// Reset Trigger to clean alarm and counter.
	
	ParamTimeRetry 			: TIME:=T#30S;				//Time to wait before a retry
	ParamNbAlms				: INT := 3;				// Parameter for the number of retries before the alarme
	ParamEnableRetryPause	: BOOL ; 
	
END_VAR

VAR_OUTPUT
	ErrorId			: UDINT;	// Error Id returned by FB ( see ADS error Code ) . 
	OUT_Completed	: BOOL ; // Reading completed successfully . 
	Busy			: BOOL ;	// FB busy to proceed command
	ModbusReadAlarm	: BOOL; 	// Alarm if three modbus attempt failed.
	
END_VAR

VAR
	R_TRIG 				: R_TRIG; 			// Rising edge detection for the trigger.
	FB_MBReadInputRegs 	: FB_MBReadInputRegs; 	// Multiple registers reading
	
	Step				: INT; 				// Grafcet step
	AlarmCounter		: INT; 				// Alarm Counter. Incremennted if modbus errOR  Alarm if counter =3 , resetable.  
	TempoRetry      		: TP;

	bRetry          		: BOOL:= FALSE; 			// Boolean to denote the retries	
	
END_VAR

// ALARM MANAGEMENT //
TempoRetry(PT := ParamTimeRetry);
	IF AlarmCounter=3 THEN 
		ModbusReadAlarm 	:=TRUE;
		bRetry := SEL(ParamEnableRetryPause , FALSE ,  TRUE);		// False = disable retry 		
	ELSE
		ModbusReadAlarm := FALSE;
		ErrorId			:= 0;
		bRetry := FALSE;		// False = disable retry 
	END_IF

OUT_Completed := FALSE ; 

// MODBUS SEQUENCE //
CASE Step OF 
	0:
		R_TRIG(CLK :=ClockRead);
		IF R_TRIG.Q THEN 
			Step :=1;
			Busy := TRUE;
		END_IF
	1:
	   FB_MBReadInputRegs(
	  			sIPAddr:= sIPAddr , 
				nTCPPort:= nTCPport ,
				nUnitID:= nUnitID,
				nQuantity:= nQuantity,
				nMBAddr:= nMBAddr, 
				cbLength:= cbLength, 
				pDestAddr:= pDestAddr, 
				bExecute:= TRUE,
				tTimeout:= tTimeout
				);
				
		IF NOT FB_MBReadInputRegs.bBusy AND NOT FB_MBReadInputRegs.bError THEN
			OUT_Completed := TRUE ;
			FB_MBReadInputRegs(bExecute:= FALSE);
			AlarmCounter	:=0; // Reset counter after successful modbus read. 
			Step 			:=0;
			Busy := FALSE;
		ELSIF NOT FB_MBReadInputRegs.bBusy AND FB_MBReadInputRegs.bError AND NOT(bRetry) THEN
			FB_MBReadInputRegs(bExecute:= FALSE);
			AlarmCounter 	:= MIN(AlarmCounter+1,3) ; 
			ErrorId			 :=FB_MBReadInputRegs.nErrId;
			Step 			:=0;
			Busy := FALSE;
		ELSIF NOT FB_MBReadInputRegs.bBusy AND FB_MBReadInputRegs.bError AND bRetry THEN
			step := 2;
			Busy := FALSE;		
			
		END_IF
	2: 
		TempoRetry(In:= TRUE);		// LEAVE SOME TIME BEFORE NEW ATTEMPT . 
		IF NOT(TempoRetry.Q) THEN
			TempoRetry(In:= FALSE);
			//AlarmCounter := 0;
			step := 0;
			
		END_IF	
END_CASE

// RESET //
	IF Reset THEN 
		AlarmCounter 		:= 0 ; 
		ErrorId 			:= 0 ; 
		ModbusReadAlarm 	:=FALSE;
		Reset 				:= FALSE;
	END_IF

// BUSY //
	//Busy 						:= FB_MBReadInputRegs.bBusy ;

ACTION Init:

END_ACTION

END_FUNCTION_BLOCK

// ---- 00_FunctionsBlocks/Communication/ModbusTCP/FB_ModbusWrite.TcPOU
FUNCTION_BLOCK FB_ModbusWrite
////////////////// 
// Write Modbus TCP/IP on Rising Edge of Trigger WriteCommAND  Returns alarm and stop modbus Read after three consecutive Modbus attempts that failed.
// Write two registers 
//////////////////
VAR_INPUT
	// Modbus ReadRegs FB inputs

	pSrcAddr			: POINTER TO BYTE ;
	sIPAddr 			: STRING(15);
	tTimeout 			: TIME;
	nTCPport			: UINT:= 502;		// TCP Port
	nMBAddr 			: WORD ;
	cbLength 			: UDINT ;
	nQuantity			: BYTE ;
	nUnitID 			: BYTE;
	WriteCmd 			: BOOL; 					// Rising Edge Trigger for sending modbus request
	
	Reset				: BOOL; 					// Reset Trigger to clean alarm and counter	
	
END_VAR


VAR_OUTPUT
	ErrorId				: UDINT; 			// Erreur ID returned by FB modbus. Updated every time on error occurs. 
	
	Completed			: BOOL ;			// Modbus Writing is completed 
	Busy				: BOOL ; 			// FB busy to proceed command
	ModbusWriteAlarm	: BOOL; 			// Alarm if three modbus attempt failed.
	
END_VAR
VAR
	R_TRIG 				: R_TRIG; 				// Rising edge detection for the trigger.
	FB_MBWriteRegs 		: FB_MBWriteRegs; 		// Multiple registers reading
	
	Step				: INT; 					// Grafcet step
	AlarmCounter		: INT; 					// Alarm Counter. Incremennted if modbus errOR  Alarm if counter =3 , resetable.  
END_VAR

Completed 				:= FALSE ;

// ALARM MANAGEMENT //
IF AlarmCounter=3 THEN
	ModbusWriteAlarm 	:=TRUE;
	
ELSE
	ModbusWriteAlarm 	:= FALSE;
	ErrorId				:= 0;
	
END_IF
	
// MODBUS SEQUENCE //
	CASE Step OF 
		0:
			R_TRIG(CLK :=WriteCmd);
			IF R_TRIG.Q THEN 
				Step :=1;
			END_IF
			
		1:
		   FB_MBWriteRegs(
					sIPAddr:= sIPAddr , 
					nTCPPort:= nTCPport ,
					nUnitID:= nUnitID,
					nQuantity:= nQuantity,
					nMBAddr:= nMBAddr, 
					cbLength:= cbLength, 
					pSrcAddr:= pSrcAddr, 
					bExecute:= TRUE,
					tTimeout:= tTimeout
					);
					
			IF NOT FB_MBWriteRegs.bBusy AND NOT FB_MBWriteRegs.bError THEN
				FB_MBWriteRegs(bExecute:= FALSE);
				AlarmCounter		:=0; // Reset counter after successful modbus read. 
				Step 				:=0;
				Completed 			:= TRUE ;
				
			ELSIF NOT FB_MBWriteRegs.bBusy AND FB_MBWriteRegs.bError THEN
				FB_MBWriteRegs(bExecute:= FALSE);
				AlarmCounter 		:=MIN(AlarmCounter+1,3) ; 
				ErrorId			 	:=FB_MBWriteRegs.nErrId;
				Step 				:=0;
				
			END_IF
			
	END_CASE

// RESET //	
	IF Reset THEN 
			AlarmCounter 	:= 0 ; 
			ErrorId 		:= 0 ; 
			Reset			:= FALSE;
	END_IF	
	
// BUSY //
	Busy 					:= FB_MBWriteRegs.bBusy ;

END_FUNCTION_BLOCK

// ---- 00_FunctionsBlocks/Communication/ModbusTCP/FB_ModbusWriteMultipleCoils.TcPOU
FUNCTION_BLOCK FB_ModbusWriteMultipleCoils
////////////////// 
// Write Modbus TCP/IP on Rising Edge of Trigger WriteCommAND  Returns alarm and stop modbus Read after three consecutive Modbus attempts that failed.
// Write two registers 
//////////////////
VAR_INPUT
	// Modbus ReadRegs FB inputs

	pSrcAddr			: POINTER TO BYTE ;
	sIPAddr 			: STRING(15);
	tTimeout 			: TIME;
	nTCPport			: UINT:= 502;		// TCP Port
	nMBAddr 			: WORD ;
	cbLength 			: UDINT ;
	nQuantity			: BYTE ;
	nUnitID 			: BYTE;
	WriteCmd 			: BOOL; 					// Rising Edge Trigger for sending modbus request
	
	Reset				: BOOL; 					// Reset Trigger to clean alarm and counter	
	
END_VAR


VAR_OUTPUT
	ErrorId				: UDINT; 			// Erreur ID returned by FB modbus. Updated every time on error occurs. 
	
	Completed			: BOOL ;			// Modbus Writing is completed 
	Busy				: BOOL ; 			// FB busy to proceed command
	ModbusWriteAlarm	: BOOL; 			// Alarm if three modbus attempt failed.
	
END_VAR
VAR
	R_TRIG 				: R_TRIG; 				// Rising edge detection for the trigger.
	FB_MBWriteCoils		: FB_MBWriteCoils; 		// Multiple registers reading
	
	Step				: INT; 					// Grafcet step
	AlarmCounter		: INT; 					// Alarm Counter. Incremennted if modbus errOR  Alarm if counter =3 , resetable.  
END_VAR

Completed 				:= FALSE ;

// ALARM MANAGEMENT //
IF AlarmCounter=3 THEN
	ModbusWriteAlarm 	:=TRUE;
	
ELSE
	ModbusWriteAlarm 	:= FALSE;
	ErrorId				:= 0;
	
END_IF
	
// MODBUS SEQUENCE //
	CASE Step OF 
		0:
			R_TRIG(CLK :=WriteCmd);
			IF R_TRIG.Q THEN 
				Step :=1;
			END_IF
			
		1:
		   FB_MBWriteCoils(
					sIPAddr:= sIPAddr , 
					nTCPPort:= nTCPport ,
					nUnitID:= nUnitID,
					nQuantity:= nQuantity,
					nMBAddr:= nMBAddr, 
					cbLength:= cbLength, 
					pSrcAddr:= pSrcAddr, 
					bExecute:= TRUE,
					tTimeout:= tTimeout
					);
					
			IF NOT FB_MBWriteCoils.bBusy AND NOT FB_MBWriteCoils.bError THEN
				FB_MBWriteCoils(bExecute:= FALSE);
				AlarmCounter		:=0; // Reset counter after successful modbus read. 
				Step 				:=0;
				Completed 			:= TRUE ;
				
			ELSIF NOT FB_MBWriteCoils.bBusy AND FB_MBWriteCoils.bError THEN
				FB_MBWriteCoils(bExecute:= FALSE);
				AlarmCounter 		:=MIN(AlarmCounter+1,3) ; 
				ErrorId			 	:=FB_MBWriteCoils.nErrId;
				Step 				:=0;
				
			END_IF
			
	END_CASE

// RESET //	
	IF Reset THEN 
			AlarmCounter 	:= 0 ; 
			ErrorId 		:= 0 ; 
	END_IF	
	
// BUSY //
	Busy 					:= FB_MBWriteCoils.bBusy ;

END_FUNCTION_BLOCK

// ---- 00_FunctionsBlocks/Communication/ModbusTCP/FB_ModbusWriteSingleCoil.TcPOU
FUNCTION_BLOCK FB_ModbusWriteSingleCoil
////////////////// 
// Write Modbus TCP/IP on Rising Edge of Trigger WriteCommAND  Returns alarm and stop modbus Read after three consecutive Modbus attempts that failed.
// Write two registers 
//////////////////
VAR_INPUT
	// Modbus ReadRegs FB inputs
	bValue 				: BOOL;
	sIPAddr 			: STRING(15);
	tTimeout 			: TIME;
	nTCPport			: UINT:= 502;		// TCP Port
	nMBAddr 			: WORD ;
	nUnitID 			: BYTE;
	WriteCmd 			: BOOL; 					// Rising Edge Trigger for sending modbus request
	
	Reset				: BOOL; 					// Reset Trigger to clean alarm and counter	
	
END_VAR


VAR_OUTPUT
	ErrorId				: UDINT; 			// Erreur ID returned by FB modbus. Updated every time on error occurs. 
	
	Completed			: BOOL ;			// Modbus Writing is completed 
	Busy				: BOOL ; 			// FB busy to proceed command
	ModbusWriteAlarm	: BOOL; 			// Alarm if three modbus attempt failed.
	
END_VAR
VAR
	R_TRIG 				: R_TRIG; 				// Rising edge detection for the trigger.
	FB_MBWriteSingleCoil: FB_MBWriteSingleCoil; 		// Multiple registers reading
	
	Step				: INT; 					// Grafcet step
	AlarmCounter		: INT; 					// Alarm Counter. Incremennted if modbus errOR  Alarm if counter =3 , resetable.  
	wValue				: WORD;
END_VAR

Completed 				:= FALSE ;

// ALARM MANAGEMENT //
IF AlarmCounter=3 THEN
	ModbusWriteAlarm 	:=TRUE;
	
ELSE
	ModbusWriteAlarm 	:= FALSE;
	ErrorId				:= 0;
	
END_IF

IF bValue THEN
	wValue := 16#FF00;
ELSE
	wValue := 16#0000;
END_IF
	
// MODBUS SEQUENCE //
	CASE Step OF 
		0:
			R_TRIG(CLK :=WriteCmd);
			IF R_TRIG.Q THEN 
				Step :=1;
			END_IF
			
		1:
		   FB_MBWriteSingleCoil
			(
				sIPAddr:= sIPAddr ,
				nValue := wValue,
				nTCPPort:= nTCPport ,
				nUnitID:= nUnitID,
				nMBAddr:= nMBAddr, 
				bExecute:= TRUE,
				tTimeout:= tTimeout
			);
					
			IF NOT FB_MBWriteSingleCoil.bBusy AND NOT FB_MBWriteSingleCoil.bError THEN
				FB_MBWriteSingleCoil(bExecute:= FALSE);
				AlarmCounter		:=0; // Reset counter after successful modbus read. 
				Step 				:=0;
				Completed 			:= TRUE ;
				
			ELSIF NOT FB_MBWriteSingleCoil.bBusy AND FB_MBWriteSingleCoil.bError THEN
				FB_MBWriteSingleCoil(bExecute:= FALSE);
				AlarmCounter 		:=MIN(AlarmCounter+1,3) ; 
				ErrorId			 	:=FB_MBWriteSingleCoil.nErrId;
				Step 				:=0;
				
			END_IF
			
	END_CASE

// RESET //	
	IF Reset THEN 
			AlarmCounter 	:= 0 ; 
			ErrorId 		:= 0 ; 
	END_IF	
	
// BUSY //
	Busy 					:= FB_MBWriteSingleCoil.bBusy ;

END_FUNCTION_BLOCK

// ---- 00_FunctionsBlocks/Communication/ModbusTCP/FB_ModbusWriteSingleRegister.TcPOU
FUNCTION_BLOCK FB_ModbusWriteSingleRegister
////////////////// 
// Write Modbus TCP/IP on Rising Edge of Trigger WriteCommAND  Returns alarm and stop modbus Read after three consecutive Modbus attempts that failed.
// Write two registers 
//////////////////
VAR_INPUT
	// Modbus ReadRegs FB inputs

	InputWord			: WORD ;
	sIPAddr 			: STRING(15);
	tTimeout 			: TIME;
	nTCPport			: UINT:= 502;		// TCP Port
	nMBAddr 			: WORD ;
	cbLength 			: UDINT ;
	nQuantity			: BYTE ;
	nUnitID 			: BYTE;
	WriteCmd 			: BOOL; 					// Rising Edge Trigger for sending modbus request
	
	Reset				: BOOL; 					// Reset Trigger to clean alarm and counter	
	
END_VAR


VAR_OUTPUT
	ErrorId						: UDINT; 			// Erreur ID returned by FB modbus. Updated every time on error occurs. 
	                    		
	Completed					: BOOL ;			// Modbus Writing is completed 
	Busy						: BOOL ; 			// FB busy to proceed command
	ModbusWriteAlarm			: BOOL; 			// Alarm if three modbus attempt failed.
	
END_VAR
VAR
	R_TRIG 						: R_TRIG; 				// Rising edge detection for the trigger.
	MBWriteSingleReg 		: FB_MBWriteSingleReg; 		// Multiple registers reading
	
	Step						: INT; 					// Grafcet step
	AlarmCounter				: INT; 					// Alarm Counter. Incremennted if modbus errOR  Alarm if counter =3 , resetable.  
END_VAR

Completed 				:= FALSE ;

// ALARM MANAGEMENT //
IF AlarmCounter=3 THEN
	ModbusWriteAlarm 	:=TRUE;
	
ELSE
	ModbusWriteAlarm 	:= FALSE;
	ErrorId				:= 0;
	
END_IF
	
// MODBUS SEQUENCE //
	CASE Step OF 
		0:
			R_TRIG(CLK :=WriteCmd);
			IF R_TRIG.Q THEN 
				Step :=1;
			END_IF
			
		1:
		   MBWriteSingleReg(
			   		nValue := InputWord,
					sIPAddr:= sIPAddr , 
					nTCPPort:= nTCPport ,
					nUnitID:= nUnitID,
					nMBAddr:= nMBAddr, 
					bExecute:= TRUE,
					tTimeout:= tTimeout
					);
					
			IF NOT MBWriteSingleReg.bBusy AND NOT MBWriteSingleReg.bError THEN
				MBWriteSingleReg(bExecute:= FALSE);
				AlarmCounter		:=0; // Reset counter after successful modbus read. 
				Step 				:=0;
				Completed 			:= TRUE ;
				
			ELSIF NOT MBWriteSingleReg.bBusy AND MBWriteSingleReg.bError THEN
				MBWriteSingleReg(bExecute:= FALSE);
				AlarmCounter 		:=MIN(AlarmCounter+1,3) ; 
				ErrorId			 	:=MBWriteSingleReg.nErrId;
				Step 				:=0;
				
			END_IF
			
	END_CASE

// RESET //	
	IF Reset THEN 
			AlarmCounter 	:= 0 ; 
			ErrorId 		:= 0 ; 
			Reset			:= FALSE;
			MBWriteSingleReg(bExecute := FALSE);
	END_IF	
	
// BUSY //
	Busy 					:= MBWriteSingleReg.bBusy ;

END_FUNCTION_BLOCK

// ---- 00_FunctionsBlocks/Ctrl/FB_PIDRegulation.TcPOU
FUNCTION_BLOCK FB_PIDRegulation
// Akuo Version of PID Regulation  for solar power plant . Input can be P or Q . 
// Out  = Error *K (1+ 1/Ti sum(error) + Td delta(error) ) 
(*
	DATE :						07/2020																										
	Developper:				GGY																												
	Version :					V1.0																										
	Function :																																																																		
*)
VAR_INPUT PERSISTENT

	ParamK				: REAL ; // Proportionnal 
	ParamTi				: REAL ; // Integral (s) . 0 to disable
	ParamTd				: REAL ; // Derivative (s). 0 to disable . 
	
	ParamXmax			: REAL ; // maximal Value for X. Shall account for number of available PTR . 
	ParamXmin			: REAL; // minimal value for X 
	
	ParamOutmax			: REAL ; // Maximal output value
	ParamOutmin			: REAL ; // Maximal input value 
	
	
	
END_VAR

VAR_INPUT
	IN_SetptX				: REAL ; // Value to reach 
	IN_MesX					: REAL ; // Measure to compare with
	IN_MesComXError			: BOOL ; // Communication lost with the measure tool. 
	IN_SetptOpenLoop		: REAL  ; // Output of the PID when disabled. This shall be equal to an evaluation of the correct output. Usually SetptX. OpenLoop setpoint. 

	
	IN_CmdReset				: BOOL ; // Reset PID 
	IN_CmdPIDOn				: BOOL ; // Activate/ Desactivate PID . outpout equals to the offset if desactivated/ 
END_VAR

VAR_OUTPUT
	OUT_X					: REAL ; // Output of the PID 
	OUT_PIDMode				: INT ; // Mode of the PID ( 1: Bypassed  , 3 : Proportionnal , 4 : PI , 5 PID , 6: PD). 
	
END_VAR
VAR
	
	CalSetptOffset 			: REAL  ; // Offset to be added to the PID to ensure continuity when resetting it or activating it. 

	IntegralX			: REAL ; // Intergal
	DerivativeX			: REAL ; // Derivative
	ErrorX				: REAL;	// Error  
	CP_PID				: BOOL;	// PID Enabled
	Clock				: TON ; // Calculate Elapsed Time ; 
	DeltaTime			: DWORD ; // 
	// Derivative
	StepDerivative		: INT := 0; // Derivative Step ( initialization , methode degre 1 , methode degre 2) 
	X2,X1				:REAL;
	T1					:DWORD;
	CalReset: BOOL;
	
	KCopy				: REAL ; 
	TiCopy				: REAL ; 
	TdCopy				: REAL ; 
	X_Temp				: REAL ; // Intermediate result . 
	
	CalOutLimitReached_Up	: BOOL;		// Output reached maximum output limit
	CalOutLimitReached_Down	: BOOL;		// Output reached minimum output limit
	
	TrigCP_PID: BOOL;
	bInit: BOOL := TRUE  ; 
	time_new: INT;
	delta_time: INT;
	time_old: INT;
END_VAR

// INITIALIZE 
	OUT_PIDMode := 1 ;

	CalReset := IN_CmdReset OR NOT IN_CmdPIDOn OR ABS(KCopy-ParamK)>0.000001 OR ABS(TiCopy-ParamTi)>0.000001 OR ABS(TdCopy-ParamTd)>0.000001 OR IN_MesComXError; // Reset if change of parameters >> passage en boucle ouverte. 

	CP_PID :=   (ParamK>0.00001 OR ParamK<-0.00001)  AND NOT CalReset  ; // PID Enable ssi Activation and K >0 and not communication alarm with power meter . and not K change . 
	

	IF NOT CP_PID OR bInit THEN 
		// Début proposition de modif KBT
		time_old := TIME_TO_INT(TIME());
		// Fin proposition de modif KBT

		
		Clock(IN:=FALSE ) ; 
		Clock(IN:=TRUE, PT:=T#1H);	//Initialize clock 
		bInit	:= FALSE ; 
	ELSE 
		Clock();
		DeltaTime	:= TIME_TO_DWORD(CLOCK.ET) ; 	// 
		
		// Début proposition de modif KBT
		time_new := TIME_TO_INT(TIME());
		IF time_old <> 0 THEN
			delta_time := time_new - time_old;
		END_IF
		time_old := TIME_TO_INT(TIME());
		// Fin proposition de modif KBT
	END_IF


	KCopy 	:=  ParamK ; 
	TiCopy	:= ParamTi ; 
	TdCopy	:= ParamTd ; 
	
// CHECK INPUT // 
	IN_SetptX := MAX(MIN(IN_SetptX, ParamXmax ), ParamXmin); // Limit the Input with Min/ Max values.

	IN_SetptOpenLoop := MAX(MIN(IN_SetptOpenLoop, ParamXmax ), ParamXmin); // Limit the Input with Min/ Max values.
	
// EVALUATE QUANTITIES //
	// Clock
	
	IF DeltaTime > 0 THEN	// We calculate on time cycle. When the time cycle is over , we reinitialize the clock
		Clock(IN:=FALSE ) ; 
		Clock(IN:=TRUE, PT:=T#1H);	//Initialize clock 
	ELSE
		CLOCK(PT:=T#1H,IN:=TRUE);
	END_IF
	// Error 
		ErrorX := IN_SetptX - IN_MesX ; 

	//Integral
		// Sauturate the integral if overflow or if limts are reached or output reaches limits Reset the integral if command reset. 
		IF (NOT(1E30 - ErrorX*DeltaTime/1000 < IntegralX OR -1E30 - ErrorX*DeltaTime/1000 > IntegralX) AND ParamTi>0 ) OR CalReset THEN
			IF NOT ((ErrorX > 0 AND  CalOutLimitReached_Up) OR (ErrorX < 0 AND CalOutLimitReached_Down)) THEN 
				IntegralX:=SEL(CalReset,IntegralX+ErrorX*DeltaTime/1000 , 0) ;
			END_IF
			
			
		END_IF
		
	// Derivative 
		IF StepDerivative=0 OR CalReset THEN		// Reinitializa derivative if reset commAND  
			X1:=ErrorX;
			X2:=ErrorX;
			T1:=DeltaTime;
			DerivativeX := 0;
			StepDerivative:=1;
		ELSIF StepDerivative=1 AND ParamTd>0 THEN 
			DerivativeX := (ErrorX - X1)/(DeltaTime-T1) ; // f'(x) = (f(x+h)-f(x))/h
			X2:=X1;
			X1:=ErrorX;
			T1:=DeltaTime;	
			StepDerivative:=2 ; 		
		ELSE	
			IF DeltaTime>0 AND DerivativeX < 1E30 AND DerivativeX> 1E30 AND ParamTd>0  THEN		// Saturate the derivative if going too high. 
				IF NOT ((ErrorX > 0 AND  CalOutLimitReached_Up) OR (ErrorX < 0 AND CalOutLimitReached_Down)) THEN 
					DerivativeX:=(3*(ErrorX)-4*X1+X2)/(2*(DeltaTime-T1)*1000);		// Formule de Gear au second degré . f'(x) = 1/2h*(3*f(x+2h)-4*f(x+h)+f(x))
					X2:=X1;
					X1:=ErrorX;
					T1:=DeltaTime;
				END_IF
			END_IF;
		END_IF;
	
// PID CALCULATION
	IF CP_PID THEN

		
		TrigCP_PID	:= TRUE ; 
		// PID Enable 
		IF  ParamTi>0 AND ParamTd>0 THEN // Integral and derivative activated
			X_Temp:=CalSetptOffset+ParamK*(ErrorX+IntegralX/ParamTi+DerivativeX*ParamTd);
			OUT_PIDMode := 5 ; 
		ELSIF ParamTd>0 THEN // Derivative activated 
			X_Temp:= CalSetptOffset+ParamK*(ErrorX+DerivativeX*ParamTd) ; 
			OUT_PIDMode := 6 ; 
		ELSIF ParamTi>0 THEN // Integral activated 
			X_Temp:=CalSetptOffset+ParamK*(ErrorX+IntegralX/ParamTi);
			OUT_PIDMode := 4 ; 
		ELSE	// Only proportionnal
			X_Temp:=CalSetptOffset+ParamK*(ErrorX) ; 
			OUT_PIDMode := 3 ; 
		END_IF
		
	ELSE
		
		CalSetptOffset := IN_SetptOpenLoop ; // At the moment when i activated the PID, i need to ensure continuity of the OUT_X and start the PID from there . 
	
		TrigCP_PID	:= FALSE ; 
		//PID Disable. Open Loop . 
		X_Temp := IN_SetptOpenLoop ;
		OUT_PIDMode:=1 ;
	END_IF
	
// Saturate the OUtput with limits : 
CalOutLimitReached_Up := (X_Temp > ParamOutmax)  ;
CalOutLimitReached_Down:= (X_Temp < ParamOutmin)  ;
 

OUT_X :=  MAX(MIN(ParamOutmax , X_Temp ) , ParamOutmin ) ;

END_FUNCTION_BLOCK

// ---- 00_FunctionsBlocks/Database/CheckConfig.TcPOU
PROGRAM CheckConfig
VAR_INPUT
		IN_Start				: BOOL := TRUE;
		ParamInitWait			: TIME := T#5S;
END_VAR
VAR_OUTPUT
		OUT_aDBConfig         		: ARRAY[0..MAX_CONFIGURATIONS] OF ST_ConfigDB;
		OUT_Busy					: BOOL;
		OUT_Error					: BOOL;
		OUT_Result					: INT;
END_VAR
VAR
	// CheckConfig    
		TON_CheckConfig				: TON;      		
		TrigCheckConfig				: R_TRIG;
		TrigInit					: F_TRIG;
		RS_CheckConfig				: RS;
		                    		
		ConfigTcDBSrvEvt  			: FB_ConfigTcDBSrvEvt(sNetId := '', tTimeout:=T#5S);
		                    		
		aAutoGrpConfig    			: ARRAY[0..MAX_CONFIGURATIONS] OF ST_ConfigAutoLogGrp;
		AX_NameBase					: ARRAY[0..MAX_CONFIGURATIONS] OF T_MaxString;
		AX_hDBID					: ARRAY[0..MAX_CONFIGURATIONS] OF BOOL;
		AX_hDBIDNull				: ARRAY[0..MAX_CONFIGURATIONS] OF BOOL;
		                    		
		nDbCount          			: UDINT;
		nAutoGrpCount     			: UDINT;

		KK : UDINT;
END_VAR

TON_CheckConfig(IN := IN_Start, PT := ParamInitWait);

TrigCheckConfig(CLK := TON_CheckConfig.Q);
RS_CheckConfig(SET := TrigCheckConfig.Q);
IF TrigCheckConfig.Q THEN
	IN_Start := FALSE;
	OUT_Result := 0;
END_IF
IF RS_CheckConfig.Q1 THEN
	
	OUT_Busy := TRUE;
	IF ConfigTcDBSrvEvt.Read(pDBConfig := ADR(OUT_aDBConfig), cbDBConfig := SIZEOF(OUT_aDBConfig), pAutologGrpConfig := ADR(aAutoGrpConfig),
			cbAutoLogGrpConfig := SIZEOF(aAutoGrpConfig),pDBCount := ADR(nDbCount),pAutoLogGrpCount := ADR(nAutoGrpCount)) THEN
		
		IF ConfigTcDBSrvEvt.bError THEN
			OUT_Result := -1;
		ELSE
			FOR KK := 0 TO MAX_CONFIGURATIONS DO
				AX_hDBID[OUT_aDBConfig[KK].hDBID] := OUT_aDBConfig[KK].hDBID <> 0;
				AX_NameBase[KK] :=  OUT_aDBConfig[KK].sName;
			END_FOR
			OUT_Result := 1;
		END_IF  
		RS_CheckConfig(RESET1 := TRUE);
		RS_CheckConfig(RESET1 := FALSE);
		OUT_Busy := FALSE;
		
	END_IF
END_IF

END_PROGRAM

// ---- 00_FunctionsBlocks/Database/Firebird/Firebird_CreateTables.TcPOU
PROGRAM Firebird_CreateTables
VAR_INPUT
	IN_Start				: BOOL;
	IN_TableNames			: ARRAY[1.. CstNbTables] OF STRING;
	IN_hDBID         		: UDINT;	
END_VAR
VAR_OUTPUT
	OUT_Error				: BOOL;
	OUT_Busy				: BOOL;
	OUT_Result				: INT;
END_VAR
VAR
	Etape					: UINT;
	
	TrigStart				: R_TRIG;
	RsStart					: RS;
	bCreateTable			: BOOL;
	TrigCreateTable			: R_TRIG;
	RsCreateTable			: RS;
	PLCDBCreateEvt 			: FB_PLCDBCreateEvt(sNetID := '', tTimeout := T#5S);
	FirebirdConf			: T_DBConfig_Odbc;
	sExtension				: STRING:= '.db';
	tcMessage    	 		: I_TcMessage;
	
	AX_ColArray				: ARRAY[0..3] OF ST_ColumnInfo;
	
	NumTable				: UINT := 1;
	KK						: UDINT;
END_VAR


AX_ColArray[0].sName := 'TimeStamp';     	AX_ColArray[0].eType := E_ColumnType.DateTime;   	AX_ColArray[0].nLength := 4;    
AX_ColArray[1].sName := 'TimeStamp_Ms';    	AX_ColArray[1].eType := E_ColumnType.Integer;    	AX_ColArray[1].nLength := 4;
AX_ColArray[2].sName := 'ParentId';   		AX_ColArray[2].eType := E_ColumnType.Integer;   	AX_ColArray[2].nLength := 4;
AX_ColArray[3].sName := 'Value';   			AX_ColArray[3].eType := E_ColumnType.Float;   		AX_ColArray[3].nLength := 8;


TrigCreateTable(CLK := IN_Start);
RsCreateTable(SET:= TrigCreateTable.Q);

IF RsCreateTable.Q1 THEN
	OUT_Busy := TRUE;
	IF NumTable <= CstNbTables THEN
		IF PLCDBCreateEvt.Table(hDBID := IN_hDBID, sTableName := IN_TableNames[NumTable],  pTableCfg := ADR(AX_ColArray), cbTableCfg := SIZEOF(AX_ColArray)  ) THEN
			IF PLCDBCreateEvt.bError THEN
				Etape := 255;
				OUT_Error := TRUE;
				OUT_Result := -2;
			ELSE
				IF Numtable = CstNbTables THEN
					IN_Start := FALSE;
					Etape := 0;
					RsCreateTable(RESET1 := TRUE);
					RsCreateTable(RESET1 := FALSE);	
					bCreateTable := FALSE;
					OUT_Result := 1;	
					TrigStart(CLK := FALSE);
					OUT_Busy := FALSE;	
					OUT_Error := FALSE;
					OUT_Result := 1;
				ELSE
					NumTable := NumTable + 1;		
				END_IF
			END_IF
		END_IF
	END_IF
END_IF

IF Etape = 255 THEN
	Etape := 0;
	bCreateTable := FALSE;
	IN_Start := FALSE;
	OUT_Busy := FALSE;	
	RsCreateTable(RESET1 := TRUE);
	RsCreateTable(RESET1 := FALSE);
END_IF

END_PROGRAM

// ---- 00_FunctionsBlocks/Database/Firebird/Firebird_InsertBuffer.TcPOU
FUNCTION_BLOCK Firebird_InsertBuffer
// Fonctionnement : Tableau de 2000 structures en input. Dès qu'on atteint 1000 structures remplies, décalage de l'espace mémoire
// pour en 1 temps de cycle pour ne pas perdre de données sur le transfert.
VAR CONSTANT
	//CstNbLigneBuffer					: UINT:= 500;
	CstNbLigneBufferMax	 				: DINT:= 1000;
                            			
END_VAR                     			
                            			
VAR_INPUT                   			
	NomTable							: STRING(255) := 'Table100ms';
	IN_Reset							: BOOL;
	IN_Hdbid							: DINT;
	ParamTimeOut						: TIME := T#10s;
END_VAR                     			
                            			
VAR_OUTPUT                  			
	OUT_Error							: BOOL;
	OUT_Busy							: BOOL;
	OUT_Result							: INT;
	Out_Connected						: BOOL;
END_VAR                     			
                            			
VAR                         		
	Etape_main							: UINT:=2;	
	ETAPE								: UINT;
		CstNbLigneBuffer					: UINT:= 500;
	FTrig_TP_Retry						: F_TRIG;                        			
	TrigReset							: R_TRIG;
	TON_Watchdog						: TON ;
	TP_Retry							: TP;
	Tmp_Nb_Buffer						: DINT;
    //myStruct      						: ARRAY[1..CstNbLigneBuffer] OF St_DataHisto;
	//myStructMax    						: ARRAY[1..CstNbLigneBufferMax] OF St_DataHisto;
	StructNull							: St_DataHisto;
                            			
    SQLDatabase1						: FB_SQLDatabaseEvt('',T#10S);
    SQLDatabase2						: FB_SQLDatabaseEvt('',T#10S);
	SQLCommand1							: FB_SQLCommandEvt('',T#10S);
	SQLCommand2							: FB_SQLCommandEvt('',T#10S);
	
	bConnected							: BOOL;              	        	
                            			
	TrameValues							: T_MaxString := ' ([Timestamp],[ParentId],[Value])';
	pPosRequete							: DINT;                		
	RequeteFinale						: ARRAY[1..10000] OF STRING(1000);	
	RequeteFinaleNull					: ARRAY [1..10000] OF STRING(1000);
	
	sTimeStamp							: STRING(255);  
	RequeteEntete						: STRING(1000);
	sInsertValue						: STRING(1000);
	Format								: FB_FormatString;
	                			
	NbElemBuffer						: DINT;
	KK									: DINT;
	                    				
	CmdStart							: BOOL;
	TrigRestartMaxReached				: R_TRIG;
	TrigCmdExec							: R_TRIG;
	TrigStart							: R_TRIG;
	RsStart								: RS;
	                        			
	// AlarmManagement      			
		bBufferMaxFull 					: BOOL;        		
		bInStructNull					: BOOL;
		
	// CONNECT	
		TrigStartConnect				: R_TRIG;	
		RsStartConnect					: RS;
	// DISCONNECT
		TrigStartDisconnect				: R_TRIG;
		RsStartDisconnect				: RS;

		bReconnect						: BOOL;
		FTrig_bReconnect				: F_TRIG;
			
	MesAlarm: BOOL;
	TrigWatchdog : R_TRIG;
	bTest: BOOL;
	FIFO						: FB_DBDatasetFifo_1min;
END_VAR    

VAR_IN_OUT
	
END_VAR


//CmdStart := FIFO.nCount>= CstNbLigneBuffer AND NOT FTrig_TP_Retry.Q;
CmdStart := FIFO.nCount >= 0 AND NOT FTrig_TP_Retry.Q;


TP_Retry(IN := FIFO.nCount >= CstNbLigneBufferMax AND NOT TP_Retry.Q, PT := T#3S);
FTrig_TP_Retry(CLK := TP_Retry.Q);

TrigReset(CLK := IN_Reset OR TON_Watchdog.Q);
IF TrigReset.Q THEN
	FIFO.A_Reset();
END_IF

TrigStart(CLK := CmdStart);
IF TrigStart.Q THEN
	ETAPE := 1;
END_IF


RsStart(SET := TrigStart.Q);
IF RsStart.Q1 THEN
	RequeteEntete :=  concat(concat(' INSERT INTO "',NomTable),'" ');
END_IF
		
CASE ETAPE OF
		
	1: // CONNECTED
		IF SQLDatabase1.CreateCmd(pSQLCommand := ADR(SQLCommand1)) THEN 
			IF NOT SQLDatabase1.bError THEN
				MEMCPY(srcAddr:= ADR(RequeteEntete), destAddr := ADR(requeteFinale), n:= SIZEOF(RequeteEntete));
				pPosRequete := LEN(STR := RequeteEntete);
				Tmp_Nb_Buffer :=UDINT_TO_DINT(FIFO.nCount -1);
				FOR KK:= 1 TO MIN(Tmp_Nb_Buffer,CstNbLigneBuffer-1) DO
					fifo.A_Get();
					sTimeStamp	:=  SYSTEMTIME_TO_STRING(fifo.Out.Timestamp);
					Format(sFormat := 'select $'%s$',%.4d,%5.2f FROM RDB$$DATABASE UNION ALL ', arg1 := F_STRING(sTimeStamp),arg2:= F_DINT(fifo.out.ParentId), arg3:= F_LREAL(fifo.out.Value), arg5:= F_STRING(NomTable), sOut=>sInsertValue);
					MEMCPY(srcAddr:= ADR(sInsertValue), destAddr := ADR(requeteFinale)+DINT_TO_DWORD(pPosRequete), n:= SIZEOF(sInsertValue));
					pPosRequete:= pPosRequete + LEN(STR := sInsertValue);
					fifo.A_Remove();
				END_FOR
				fifo.A_Get();
				sTimeStamp	:= SYSTEMTIME_TO_STRING(fifo.Out.Timestamp);
				Format(sFormat := 'select $'%s$',%.4d,%5.2f FROM RDB$$DATABASE;', arg1 := F_STRING(sTimeStamp),arg2:= F_DINT(fifo.out.ParentId), arg3:= F_LREAL(fifo.out.Value), sOut=>sInsertValue);
				MEMCPY(srcAddr:= ADR(sInsertValue), destAddr := ADR(requeteFinale)+DINT_TO_DWORD(pPosRequete), n:= SIZEOF(sInsertValue));
				fifo.A_Remove();
				IF Tmp_Nb_Buffer > 0 THEN
					ETAPE := Etape_main;
				END_IF
			ELSIF SQLDatabase1.bError THEN
				ETAPE := 255;
			END_IF
		END_IF
	2:

		IF SQLCommand1.Execute(pSQLCmd := ADR(RequeteFinale), cbSQLCmd := SIZEOF(Requetefinale))THEN
			
			IF  NOT SQLCommand1.bError THEN
				ETAPE := 4;
			ELSIF SQLCommand1.bError THEN
				ETAPE := 255;
			END_IF
		END_IF

	4:
		IF NOT SQLDatabase1.bError THEN
			
			RequeteFinale := RequeteFinaleNull;
			
			//RequeteFinale := '';
			Tmp_Nb_Buffer := MIN(UDINT_TO_DINT(FIFO.nCount),CstNbLigneBuffer);
			//FOR KK:= 1 TO Tmp_Nb_Buffer DO
			//	fifo.A_Remove();
			//END_FOR
			TrigStart(CLK := FALSE);
			RsStart(RESET1 := TRUE);
			RsStart(RESET1 := FALSE);
			TrigCmdExec(CLK := FALSE);
			CmdStart := FALSE;
			Etape := 0;
			OUT_Error := FALSE;
		ELSE 
			ETAPE := 255;
		END_IF
	255: 
		RequeteFinale := RequeteFinaleNull;

		SQLCommand1 := SQLCommand2;
		SQLDatabase1 := SQLDatabase2;
		OUT_Error := TRUE;
		RsStart(RESET1 := TRUE);
		RsStart(RESET1 := FALSE);
		TrigCmdExec(CLK := FALSE);
		CmdStart := FALSE;
		ETAPE := 0;
END_CASE

METHOD M_AddLine : BOOL
VAR_INPUT
	InStruct			: St_DataHisto;
END_VAR

VAR
	InsStruct: St_DataHisto;
END_VAR
fifo.in := InStruct;
fifo.A_Add();
END_METHOD

METHOD M_AlarmManager : BOOL
VAR_INPUT
	AlarmCode : WORD;
	
END_VAR


AlarmCode.0 := bBufferMaxFull;
AlarmCode.1 := bInStructNull;
END_METHOD

METHOD M_Connect : BOOL

VAR_OUTPUT
END_VAR
VAR_INPUT
	IN_hDBID				: DINT;
	IN_Start				: BOOL;
END_VAR
TrigStartConnect(CLK := IN_Start);
RsStartConnect(SET := TrigStartConnect.Q);
IF RsStartConnect.Q1 THEN
	IF SQLDatabase1.Connect(hDBID := IN_hDBID) THEN;
		RsStartConnect(RESET1 := TRUE);
		RsStartConnect(RESET1 := FALSE);
		bReconnect := FALSE;
	END_IF
END_IF

Out_Connected := SQLDatabase1.bConnected;
END_METHOD

METHOD M_Disconnect : BOOL
VAR_INPUT
END_VAR
VAR_INPUT
	IN_Start				: BOOL;
END_VAR
TrigStartDisconnect(CLK := IN_Start);
RsStartDisconnect(SET := TrigStartDisconnect.Q);
IF RsStartDisconnect.Q1 THEN
	FIFO.A_Reset();
	IF SQLDatabase1.Disconnect() THEN;
		RsStartDisconnect(RESET1 := TRUE);
		RsStartDisconnect(RESET1 := FALSE);
	END_IF
END_IF

Out_Connected := SQLDatabase1.bConnected;
END_METHOD

METHOD M_Init

VAR
	LL	: SINT;
	KK 	: SINT;
END_VAR
//Initialisation BUFFER
	//Buffer pour la lecture des sms
	FIFO.A_Reset();
	FIFO.A_Add();
	FIFO.A_Get();
	FIFO.A_Remove();
END_METHOD

END_FUNCTION_BLOCK

// ---- 00_FunctionsBlocks/Fifo/FB_DBDatasetFifo_1min.TcPOU
FUNCTION_BLOCK FB_DBDatasetFifo_1min
VAR_INPUT
    bOverwrite : BOOL;
    In         : St_DataHisto_Epoch;
END_VAR
VAR_OUTPUT
    bOk        : BOOL;
    nCount     : UDINT;
    nLoad      : UDINT;
    Out        : St_DataHisto_Epoch;
END_VAR
VAR
    arrBuffer  : ARRAY[0..Max_buffer_size_G] OF BYTE; (* Buffer memory used by FB_MemRingBuffer function block *)
    fbBuffer   : FB_MemRingBuffer;
END_VAR

ACTION A_Add:
fbBuffer.A_AddTail(pWrite := ADR(in),
						   cbWrite:=SIZEOF(in),
						   pBuffer:=ADR(arrBuffer),
						   cbBuffer:=SIZEOF(arrBuffer),
						   bOK=>bOK,
						   nCount =>nCount);
IF NOT bOK THEN 
	IF bOverwrite THEN
		fbBuffer.A_RemoveHead();(*remove one oldest entry*)
		fbBuffer.A_AddTail(bOK => bOk,nCount => nCount);
	END_IF
END_IF

nload := (fbbuffer.cbSize * 100)/(Max_buffer_size_G);
END_ACTION

ACTION A_Get:
fbBuffer.A_GetHead(pWrite := ADR(out),
						   cbWrite:=SIZEOF(out),
						   pBuffer:=ADR(arrBuffer),
						   cbBuffer:=SIZEOF(arrBuffer),
						   bOK=>bOK,
						   nCount =>nCount);
nload := (fbbuffer.cbSize * 100)/(Max_buffer_size_G);
END_ACTION

ACTION A_Remove:
fbBuffer.A_RemoveHead(pRead:=ADR(out),
						cbRead:=SIZEOF(out),
						pBuffer:=ADR(arrBuffer),
						cbBuffer:=SIZEOF(arrBuffer),
						bOK=>bOK,
						nCount =>nCount);
nload := (fbbuffer.cbSize * 100)/(Max_buffer_size_G);
END_ACTION

ACTION A_Reset:
MEMSET(ADR(arrBuffer),0,SIZEOF(arrBuffer)); (*reset internal buffer*)
fbBuffer.A_Reset(bOK=>bOK,nCount=>ncount);
nload := (fbbuffer.cbSize * 100)/(Max_buffer_size_G);
END_ACTION

END_FUNCTION_BLOCK

// ---- 00_FunctionsBlocks/Database/Firebird/Firebird_InsertBuffer_vEpoch.TcPOU
FUNCTION_BLOCK Firebird_InsertBuffer_vEpoch
// Fonctionnement : Tableau de 2000 structures en input. Dès qu'on atteint 1000 structures remplies, décalage de l'espace mémoire
// pour en 1 temps de cycle pour ne pas perdre de données sur le transfert.
VAR CONSTANT
	//CstNbLigneBuffer					: UINT:= 500;
	CstNbLigneBufferMax	 				: DINT:= 1000;
                            			
END_VAR                     			
                            			
VAR_INPUT                   			
	NomTable							: STRING(255) := 'Table100ms';
	IN_Reset							: BOOL;
	IN_Hdbid							: DINT;
	ParamTimeOut						: TIME := T#10s;
END_VAR                     			
                            			
VAR_OUTPUT                  			
	OUT_Error							: BOOL;
	OUT_Busy							: BOOL;
	OUT_Result							: INT;
	OUT_Connected						: BOOL;
END_VAR                     			
                            			
VAR                         			
	ETAPE								: UINT;
	CstNbLigneBuffer					: UINT:= 250;
	
	FTrig_TP_Retry						: F_TRIG;                        			
	TrigReset							: R_TRIG;
	TON_Watchdog						: TON ;
	TP_Retry							: TP;
	Tmp_Nb_Buffer						: DINT;
	StructNull							: St_DataHisto;
                            			
    SQLDatabase1						: FB_SQLDatabaseEvt('',T#10S);
    SQLDatabase2						: FB_SQLDatabaseEvt('',T#10S);
	SQLCommand1							: FB_SQLCommandEvt('',T#10S);
	SQLCommand2							: FB_SQLCommandEvt('',T#10S);
	
	bConnected							: BOOL;              	        	
                            			
	TrameValues							: T_MaxString := ' ([Timestamp],[ParentId],[Value])';
	pPosRequete							: DINT;                		
	RequeteFinale						: ARRAY[1..1000] OF STRING(1000);	
	RequeteFinaleNull					: ARRAY [1..1000] OF STRING(1000);
	
	sTimeStamp							: STRING(255);  
	RequeteEntete						: STRING(1000);
	sInsertValue						: STRING(1000);
	Format								: FB_FormatString;
	                			
	NbElemBuffer						: DINT;
	KK									: DINT;
	                    				
	CmdStart							: BOOL;
	TrigRestartMaxReached				: R_TRIG;
	TrigCmdExec							: R_TRIG;
	TrigStart							: R_TRIG;
	RsStart								: RS;
	                        			
	// AlarmManagement      			
		bBufferMaxFull 					: BOOL;        		
		bInStructNull					: BOOL;
		
	// CONNECT	
		TrigStartConnect				: R_TRIG;	
		RsStartConnect					: RS;
	// DISCONNECT
		TrigStartDisconnect				: R_TRIG;
		RsStartDisconnect				: RS;

		bReconnect						: BOOL;
		FTrig_bReconnect				: F_TRIG;
			
	MesAlarm: BOOL;
	TrigWatchdog : R_TRIG;
	bTest: BOOL;
	FIFO						: FB_DBDatasetFifo_1min;
END_VAR    

VAR_IN_OUT
	
END_VAR


//CmdStart := FIFO.nCount>= CstNbLigneBuffer AND NOT FTrig_TP_Retry.Q;
CmdStart := FIFO.nCount > 0 ;//AND NOT FTrig_TP_Retry.Q;


TP_Retry(IN := FIFO.nCount >= CstNbLigneBufferMax AND NOT TP_Retry.Q, PT := T#3S);
FTrig_TP_Retry(CLK := TP_Retry.Q);

TrigReset(CLK := IN_Reset OR TON_Watchdog.Q);
IF TrigReset.Q THEN
	FIFO.A_Reset();
	cmdStart := FALSE;
END_IF

TrigStart(CLK := CmdStart);
IF TrigStart.Q THEN
	ETAPE := 1;
END_IF


RsStart(SET := TrigStart.Q);
IF RsStart.Q1 THEN
	RequeteEntete :=  concat(concat(' INSERT INTO "',NomTable),'" ');
END_IF
		
CASE ETAPE OF
		
	1: // CONNECTED
		OUT_Busy := TRUE;
		IF SQLDatabase1.CreateCmd(pSQLCommand := ADR(SQLCommand1)) THEN 
			IF NOT SQLDatabase1.bError THEN
				MEMCPY(srcAddr:= ADR(RequeteEntete), destAddr := ADR(requeteFinale), n:= SIZEOF(RequeteEntete));
				pPosRequete := LEN(STR := RequeteEntete);
				Tmp_Nb_Buffer :=UDINT_TO_DINT(FIFO.nCount -1);
				FOR KK:= 1 TO MIN(Tmp_Nb_Buffer,CstNbLigneBuffer-1) DO
					fifo.A_Get();
					sTimeStamp	:=  ULINT_TO_STRING(fifo.Out.Timestamp);
					Format(sFormat := 'select $'%s$',%d,%5.2f FROM RDB$$DATABASE UNION ALL ', arg1 := F_STRING(sTimeStamp),arg2:= F_DINT(fifo.out.ParentId), arg3:= F_LREAL(fifo.out.Value), arg5:= F_STRING(NomTable), sOut=>sInsertValue);
					MEMCPY(srcAddr:= ADR(sInsertValue), destAddr := ADR(requeteFinale)+DINT_TO_DWORD(pPosRequete), n:= SIZEOF(sInsertValue));
					pPosRequete:= pPosRequete + LEN(STR := sInsertValue);
					fifo.A_Remove();
				END_FOR
				fifo.A_Get();
				sTimeStamp	:=  ULINT_TO_STRING(fifo.Out.Timestamp);
				Format(sFormat := 'select $'%s$',%d,%5.2f FROM RDB$$DATABASE;', arg1 := F_STRING(sTimeStamp),arg2:= F_DINT(fifo.out.ParentId), arg3:= F_LREAL(fifo.out.Value), sOut=>sInsertValue);
				MEMCPY(srcAddr:= ADR(sInsertValue), destAddr := ADR(requeteFinale)+DINT_TO_DWORD(pPosRequete), n:= SIZEOF(sInsertValue));
				fifo.A_Remove();
				IF Tmp_Nb_Buffer > 0 THEN
					ETAPE := 2;
				END_IF
			ELSIF SQLDatabase1.bError THEN
				ETAPE := 255;
			END_IF
		END_IF
	2:

		IF SQLCommand1.Execute(pSQLCmd := ADR(RequeteFinale), cbSQLCmd := SIZEOF(Requetefinale))THEN
			
			IF  NOT SQLCommand1.bError THEN
				ETAPE := 4;
			ELSIF SQLCommand1.bError THEN
				ETAPE := 255;
			END_IF
		END_IF

	4:
		IF NOT SQLDatabase1.bError THEN
			
			RequeteFinale := RequeteFinaleNull;
			
			//RequeteFinale := '';
			Tmp_Nb_Buffer := MIN(UDINT_TO_DINT(FIFO.nCount),CstNbLigneBuffer);
			//FOR KK:= 1 TO Tmp_Nb_Buffer DO
			//	fifo.A_Remove();
			//END_FOR
			TrigStart(CLK := FALSE);
			RsStart(RESET1 := TRUE);
			RsStart(RESET1 := FALSE);
			TrigCmdExec(CLK := FALSE);
			CmdStart := FALSE;
			Etape := 0;
			OUT_Error := FALSE;
			OUT_Busy := FALSE;

		ELSE 
			ETAPE := 255;
		END_IF
	255: 
		RequeteFinale := RequeteFinaleNull;

		SQLCommand1 := SQLCommand2;
		SQLDatabase1 := SQLDatabase2;
		OUT_Error := TRUE;
		RsStart(RESET1 := TRUE);
		RsStart(RESET1 := FALSE);
		TrigCmdExec(CLK := FALSE);
		CmdStart := FALSE;
		ETAPE := 0;
		OUT_Busy := FALSE;
END_CASE

METHOD M_AddLine : BOOL
VAR_INPUT
	InStruct			: St_DataHisto_Epoch;
END_VAR

VAR
END_VAR
fifo.in := InStruct;
fifo.A_Add();
END_METHOD

METHOD M_AlarmManager : BOOL
VAR_INPUT
	AlarmCode : WORD;
	
END_VAR


AlarmCode.0 := bBufferMaxFull;
AlarmCode.1 := bInStructNull;
END_METHOD

METHOD M_Connect : BOOL

VAR_OUTPUT
END_VAR
VAR_INPUT
	IN_hDBID				: DINT;
	IN_Start				: BOOL;
END_VAR
TrigStartConnect(CLK := IN_Start);
RsStartConnect(SET := TrigStartConnect.Q);
IF RsStartConnect.Q1 THEN
	IF SQLDatabase1.Connect(hDBID := IN_hDBID) THEN;
		RsStartConnect(RESET1 := TRUE);
		RsStartConnect(RESET1 := FALSE);
		bReconnect := FALSE;
	END_IF
END_IF

Out_Connected := SQLDatabase1.bConnected;
IF NOT OUT_Connected THEN
	btest := TRUE;
	
END_IF
END_METHOD

METHOD M_Disconnect : BOOL
VAR_INPUT
END_VAR
VAR_INPUT
	IN_Start				: BOOL;
END_VAR
TrigStartDisconnect(CLK := IN_Start);
RsStartDisconnect(SET := TrigStartDisconnect.Q);
IF RsStartDisconnect.Q1 THEN
	IF SQLDatabase1.Disconnect() THEN;
		RsStartDisconnect(RESET1 := TRUE);
		RsStartDisconnect(RESET1 := FALSE);
	END_IF
END_IF

Out_Connected := SQLDatabase1.bConnected;
END_METHOD

METHOD M_Init

VAR
	LL	: SINT;
	KK 	: SINT;
END_VAR
//Initialisation BUFFER
	//Buffer pour la lecture des sms
	FIFO.A_Reset();
	FIFO.A_Add();
	FIFO.A_Get();
	FIFO.A_Remove();
END_METHOD

END_FUNCTION_BLOCK

// ---- 00_FunctionsBlocks/Database/Firebird/Firebird_ReadAlarms.TcPOU
PROGRAM Firebird_ReadAlarms
VAR_INPUT
	ParamTimeBetweenReconnect	: TIME := T#1M;
	IN_StartRead				: BOOL;
	IN_FrequencyRead			: TIME := T#1M;
	IN_bAct						: BOOL; // Read only Active values
	IN_FilterAct				: BOOL;
	IN_bAck						: BOOL; // Read only Acknowledged values
	IN_FilterAck				: BOOL;
	
	IN_TimeStampStart			: TIMESTRUCT;
	IN_TimeStampEnd				: TIMESTRUCT;
	
END_VAR
VAR CONSTANT
	NbMaxElements	 			: UINT := 250;
END_VAR
VAR_OUTPUT
	OUT_Busy					: BOOL;
	
END_VAR
VAR
	
	AX_Buffer_Alarms			: ARRAY[1..NbMaxElements] OF St_AlarmsV2;		// Buffer of alarms to write
	StNull						: St_AlarmsV2;		// Buffer of alarms to write
		
	// Connexion
		TP_Reconnect			: TP;
		Trig_Connect			: R_TRIG;
		TRIG_CmdStart			: R_TRIG;
		RS_Connect				: RS;
		RS_HasBeenConnected		: RS;
	// DISCONNECT
		TrigStartDisconnect				: R_TRIG;
		RsStartDisconnect				: RS;		
			
	// READ File       
		TP_ReadBddPeriodically	: TP;
		TRIG_ReadBddPeriodically: R_TRIG;

		ETAPE					: UINT;
		Trig_Start				: R_TRIG;   
		RS_Start				: RS; 	
		Requete					: ARRAY[1..10] OF STRING(1000);
		RequeteNull				: ARRAY[1..10] OF STRING(1000);
		sToAdd					: STRING(1000);
		pPosRequete				: DINT;
		TimeStampNull			: TIMESTRUCT;
		TimeStampDefault		: TIMESTRUCT;
		sTimeStampStart			: STRING(255);
		sTimeStampEnd			: STRING(255);
		sValue					: STRING(255);
		sAck					: STRING(255);
		Format					: FB_FormatString;
		SQLDatabase				: FB_SQLDatabaseEvt('',T#10S);
		SQLCommand				: FB_SQLCommandEvt('',T#10S);
		SQLCommandNull			: FB_SQLCommandEvt('',T#10S);
		SQLResult				: FB_SQLResultEvt('',T#10S);
		
	
	// General variables
		nbMax					: UINT;
		bInit 					: BOOL;
		NomTableAlarms			: STRING(255) := 'TABLE_ALARMS_V2';
		KK						: UINT;
		
	//TABLEAU
	
		AX_MesAlarmCode_Bool	: ARRAY [1..CstNbAlarmCode] OF ARRAY[1..15] OF BOOL; //Tableau de tous les alarmesCode en Bool
		AX_Alarm_State			: ARRAY [1..CstNbAlarmCode] OF ARRAY[1..15] OF BOOL; //Tableau de Bool avec toutes les nouveaux bit modifiés
		AX_MesAck				: ARRAY [1..CstNbAlarmCode] OF ARRAY[1..15] OF BOOL;
		AX_Ack_State			: ARRAY [1..CstNbAlarmCode] OF ARRAY[1..15] OF BOOL; //Tableau de Bool avec tous les nouveaux acknowledgement 

	

END_VAR

// DataProcessing
IF NOT bInit THEN
	M_Init();
END_IF
RS_HasBeenConnected(SET := SQLDatabase.bConnected);
TP_Reconnect(In :=RS_HasBeenConnected.Q1 AND NOT SQLDatabase.bConnected OR NOT bInit OR TP_Reconnect.Q, PT := ParamTimeBetweenReconnect);
	
TP_ReadBddPeriodically(IN := NOT TP_ReadBddPeriodically.Q, PT := IN_FrequencyRead);
TRIG_ReadBddPeriodically(CLK := TP_ReadBddPeriodically.Q);
TRIG_CmdStart(CLK := IN_StartRead);

Trig_Start(CLK := SQLDatabase.bConnected AND NOT OUT_Busy AND ( TRIG_CmdStart.Q OR TRIG_ReadBddPeriodically.Q));
IF Trig_Start.Q THEN
	// Init the table :
	FOR KK := 1 TO 10 DO 
		Requete[KK] := RequeteNull[KK];
	END_FOR
	FOR KK := 1 TO NbMaxElements DO
		AX_Buffer_Alarms[KK] := StNull;
	END_FOR
	Requete := RequeteNull;
	nbMax := NbMaxElements;
	pPosRequete := 0;
	// Je commence par préparer ma requête 
	IF MEMCMP(pBuf1 := ADR(IN_TimeStampStart), pBuf2:=ADR(TimeStampNull), n:=SIZEOF(TimeStampNull))=0 THEN
		IN_TimeStampStart := TimeStampDefault;
	END_IF
	sTimeStampStart := systemtime_to_string(in := IN_TimeStampStart);
	sTimeStampEnd := systemtime_to_string(in := IN_TimeStampEnd);
	Format( sFormat := 'Select first %d "TIMESTAMP_START", case when "TIMESTAMP_STOP" is null then cast($'01.01.1970, 00:00:00.000$' as timestamp) else "TIMESTAMP_STOP" end,AlarmsID,Act,Ack from %s where "TIMESTAMP_START" > $'%s$' ', 
		sOut=> sToAdd,
		arg1 := F_UINT(In:=nbMax),
		arg2 := F_STRING(In := NomTableAlarms),
		arg3 := F_STRING(in := sTimeStampStart)
	);
	MEMCPY(destAddr := ADR(requete), srcAddr := ADR(sToAdd), n := SIZEOF(sToAdd));
	pPosRequete:= pPosRequete + LEN(STR := sToAdd);
	
	IF IN_FilterAct THEN
		sToAdd := CONCAT(STR1 := ' AND Act = ', STR2 := UINT_TO_STRING(BOOL_TO_UINT(IN_bAct)));
		MEMCPY(srcAddr:= ADR(sToAdd), destAddr := ADR(Requete)+DINT_TO_DWORD(pPosRequete), n:= SIZEOF(sToAdd));
		pPosRequete:= pPosRequete + LEN(STR := sToAdd);
	END_IF
	
	IF IN_FilterAck THEN
		sToAdd := CONCAT(STR1 := ' AND Ack = ', STR2 := UINT_TO_STRING(BOOL_TO_UINT(IN_bAck)));
		MEMCPY(srcAddr:= ADR(sToAdd), destAddr := ADR(Requete)+DINT_TO_DWORD(pPosRequete), n:= SIZEOF(sToAdd));
		pPosRequete:= pPosRequete + LEN(STR := sToAdd);
	END_IF	

	sToAdd := ' order by TIMESTAMP_START desc';
	MEMCPY(srcAddr:= ADR(sToAdd), destAddr := ADR(Requete)+DINT_TO_DWORD(pPosRequete), n:= SIZEOF(sToAdd));
	pPosRequete:= pPosRequete + LEN(STR := sToAdd);	
	ETAPE := 1;
END_IF
		
CASE ETAPE OF
	1: // CONNECTED
		OUT_Busy := TRUE;
		IF SQLDatabase.CreateCmd(pSQLCommand := ADR(SQLCommand)) THEN 
			IF NOT SQLCommAND bError THEN
				ETAPE := 2;
			ELSIF SQLCommAND bError THEN
				ETAPE := 255;
			END_IF
		END_IF
		
	2:	
		IF SQLCommAND ExecuteDataReturn(pSQLCmd := ADR(Requete), cbSQLCmd := SIZEOF(Requete), pSQLDBResult := ADR(SQLResult))THEN
			IF  NOT SQLCommAND bError THEN
				ETAPE := 3;
			ELSIF SQLCommAND bError THEN
				ETAPE := 255;
			END_IF
		END_IF
	3: 
		IF SQLResult.Read(nStartIndex := 1, nRecordCount := NbMaxElements, pData := ADR(AX_Buffer_Alarms), cbData := SIZEOF(AX_Buffer_Alarms), bDataRelease := TRUE, bWithVerifying := FALSE) THEN
			IF NOT SQLResult.bError THEN
				Etape := 4;
			ELSE
				ETAPE := 255;
			END_IF
		END_IF
	4:
		IF NOT SQLDatabase.bError THEN

			Requete  := RequeteNull;
			Trig_Start(CLK := FALSE);
			Etape := 0;
			OUT_Busy := FALSE;
		ELSE 
			ETAPE := 255;
		END_IF
	255: 
		OUT_Busy := FALSE;
		Requete := RequeteNull;
		Etape := 0;
		IN_StartRead := FALSE;
END_CASE

METHOD M_Connect : BOOL

VAR_OUTPUT
END_VAR
VAR_INPUT
	IN_hDBID				: DINT;
	IN_Start				: BOOL;
END_VAR
Trig_Connect(CLK := IN_Start);
RS_Connect(SET := Trig_Connect.Q);
IF RS_Connect.Q1 THEN
	IF SQLDatabase.Connect(hDBID := IN_hDBID) THEN;
		RS_Connect(RESET1 := TRUE);
		RS_Connect(RESET1 := FALSE);
	END_IF
END_IF
END_METHOD

METHOD M_Disconnect : BOOL
VAR_INPUT
END_VAR
VAR_INPUT
	IN_Start				: BOOL;
END_VAR
TrigStartDisconnect(CLK := IN_Start);
RsStartDisconnect(SET := TrigStartDisconnect.Q);
IF RsStartDisconnect.Q1 THEN
	IF SQLDatabase.Disconnect() THEN;
		RsStartDisconnect(RESET1 := TRUE);
		RsStartDisconnect(RESET1 := FALSE);
	END_IF
END_IF
END_METHOD

METHOD M_Init

VAR
	LL	: SINT;
	KK 	: SINT;
END_VAR
TimeStampDefault.wYear := 1995;
TimeStampDefault.wMonth := 3;
TimeStampDefault.wDay := 12;

bInit := TRUE;
END_METHOD

END_PROGRAM

// ---- 00_FunctionsBlocks/Database/Firebird/Firebird_RetrieveHDBID.TcPOU
PROGRAM Firebird_RetrieveHDBID
VAR_INPUT
	IN_ConfigDbActuelle		: ARRAY[0..MAX_CONFIGURATIONS] OF ST_ConfigDB; 
	IN_Dir					: T_MAXSTRING;
	IN_Name					: ARRAY[1..CstNbBases] OF STRING;
	IN_Start				: BOOL;
	IN_IpAddressServer		: STRING := 'localhost';
	IN_Port					: STRING := '3050';
END_VAR

VAR_OUTPUT
	OUT_hDBID         		: ARRAY[1..CstNbBases] OF DINT;	
	OUT_Error				: BOOL;
	OUT_Busy				: BOOL;
	OUT_Result				: INT;
END_VAR
VAR
	TrigStart				: R_TRIG;
	KK 						: UDINT;
	sExtension				: STRING;
	DbFullDirName			:  ARRAY[1..CstNbBases] OF STRING;
	LL						: DINT := 1;
	RS_Start				: RS;
END_VAR


sExtension := '.FDB';
FOR KK := 1 TO CstNbBases DO
	DbFullDirName[KK] := CONCAT(str1:= IN_IpAddressServer, STR2:= CONCAT(str1:= '/',str2:= CONCAT(STR1:= IN_Port, str2:=concat(str1 := ':', str2:=Concat(STR1:=Concat(STR1:= IN_Dir, STR2 := IN_Name[KK]), STR2 := sExtension)))));
END_FOR
TrigStart(CLK := IN_Start );
IF TrigStart.Q THEN
	LL := 1;
END_IF
RS_Start(SET := TrigStart.Q);
IF RS_Start.Q1 THEN

	OUT_Busy := TRUE;
	IF LL <= CstNbBases AND LL >0 THEN
		FOR KK := 0 TO MAX_CONFIGURATIONS DO
			IF IN_ConfigDbActuelle[KK].sDatabase = DbFullDirName[LL] THEN
				OUT_hDBID[LL] := IN_ConfigDbActuelle[KK].hDBID;
				LL := LL+1;
				EXIT;
			END_IF
			IF KK = MAX_CONFIGURATIONS THEN
				OUT_Result := -2;
				LL := -2;
				OUT_Error := TRUE;
				OUT_Busy := FALSE;
			END_IF
		END_FOR
	ELSIF LL > CstNbBases THEN
		OUT_Result := 1;
		OUT_Busy := FALSE;
		OUT_Error := FALSE;
		LL := 1;
		RS_Start(RESET1 := TRUE);
		RS_Start(RESET1 := FALSE);
	END_IF
END_IF

END_PROGRAM

// ---- 00_FunctionsBlocks/Database/Firebird/Firebird_SelectBuffer.TcPOU
FUNCTION_BLOCK Firebird_SelectBuffer
VAR CONSTANT
	CstNbLigne							: DINT:= 250;
                            			
END_VAR                     			
                            			
VAR_INPUT                   			
	IN_NomTable							: STRING := 'Table100ms';
	IN_IdToSelect						: UINT;
	IN_TimeStampStart					: TIMESTRUCT;
	IN_hDBID							: UDINT;
	IN_Reset							: BOOL;
	IN_Start							: BOOL;
END_VAR  
VAR_OUTPUT                  			
	OUT_Error							: BOOL;
	OUT_Busy							: BOOL;
	OUT_Result							: INT;
	Out_Connected						: BOOL;
	Out_Array							: ARRAY[1..CstNbLigne] OF St_DataHisto;
END_VAR 

VAR                         			
	ETAPE								: UINT;
	NbLigne								: DINT;                        			
	TrigReset							: R_TRIG;
	
	StringTimeStart						: STRING;
		                    			
	StructNull							: St_DataHisto;
                            			
    SQLDatabase							: FB_SQLDatabaseEvt('',T#10S);
	SQLCommand							: FB_SQLCommandEvt('',T#10S);
	SQLCommandNull						: FB_SQLCommandEvt('',T#10S);
	SQLResult	 						: FB_SQLResultEvt(sNetID:='', tTimeout   := T#5S); 
	bConnected							: BOOL;              	        	
                            			
	pPosRequete							: DINT;                		
	RequeteFinale						: STRING(1000);	
	RequeteFinaleNull					: STRING(1000);	
	sTimeStamp							: STRING(255);  
	Format								: FB_FormatString;
	                			
	KK									: DINT;
	                    				
	CmdStart							: BOOL;
	TrigCmdExec							: R_TRIG;
	TrigStart							: R_TRIG;
	RsStart								: RS;
	                        			
	// AlarmManagement      			
		bBufferMaxFull 					: BOOL;        		
		bInStructNull					: BOOL;
		
	// CONNECT	
		TrigStartConnect				: R_TRIG;	
		RsStartConnect					: RS;
END_VAR

TrigReset(CLK := IN_Reset);
IF TrigReset.Q THEN

	//SQLCommand := SQLCommandNull;
END_IF

TrigStart(CLK := IN_Start);
IF TrigStart.Q THEN
	NbLigne := CstNbLigne;
	StringTimeStart := LEFT(STR := SYSTEMTIME_TO_STRING(IN_TimeStampStart), SIZE := LEN(SYSTEMTIME_TO_STRING(IN_TimeStampStart))-4);
	
	Format(sFormat := 'Select first %d * from "%s" where "ParentId" = %d and "TimeStamp" > $'%s$'', sOut => RequeteFinale, 
	arg1 := F_DINT(in := NbLigne), arg2 := F_STRING(in := IN_NomTable), arg3 := F_UINT(in := IN_IdToSelect), arg4:= F_STRING(in := StringTimeStart));
	ETAPE := 1;
END_IF

CASE ETAPE OF
		
	1: // CONNECTED
		IF SQLDatabase.CreateCmd(pSQLCommand := ADR(SQLCommand)) THEN 
			IF NOT SQLCommAND bError THEN
				ETAPE := 2;
			ELSIF SQLCommAND bError THEN
				ETAPE := 255;
			END_IF
		END_IF
	2:
		
		IF SQLCommAND ExecuteDataReturn(pSQLCmd := ADR(RequeteFinale), cbSQLCmd := SIZEOF(RequeteFinale), pSQLDBResult := ADR(SQLResult)) THEN
    		IF SQLCommAND bError THEN
    		    ETAPE := 255; 
    		ELSE
    		    ETAPE := 3; 
    		END_IF			
		END_IF
	3:
		IF SQLResult.Read(nStartIndex := 0, nRecordCount := CstNbLigne, pData := ADR(Out_Array), cbData := SIZEOF(Out_Array), bWithVerifying := TRUE, bDataRelease:= TRUE) THEN
			IF NOT SQLResult.bError THEN
				ETAPE := 4;
			ELSE
				ETAPE := 255;
			END_IF
		END_IF
		
	4:
		IF NOT SQLDatabase.bError THEN
			
			RequeteFinale := RequeteFinaleNull;
	
			TrigStart(CLK := FALSE);
			RsStart(RESET1 := TRUE);
			RsStart(RESET1 := FALSE);
			TrigCmdExec(CLK := FALSE);
			IN_Start := FALSE;
			Etape := 0;
			OUT_Error := FALSE;
		ELSE 
			ETAPE := 255;
		END_IF
	255: 
		RequeteFinale := RequeteFinaleNull;
		//RequeteFinale := '';
		OUT_Error := TRUE;
		Etape := 0;
		RsStart(RESET1 := TRUE);
		RsStart(RESET1 := FALSE);
		TrigCmdExec(CLK := FALSE);
		IN_Start := FALSE;
END_CASE

METHOD M_Connect : BOOL

VAR_OUTPUT
END_VAR
VAR_INPUT
	IN_hDBID				: UDINT;
	IN_Start				: BOOL;
END_VAR
TrigStartConnect(CLK := IN_Start);
RsStartConnect(SET := TrigStartConnect.Q);
IF RsStartConnect.Q1 THEN
	IF SQLDatabase.Connect(hDBID := IN_hDBID) THEN;
		RsStartConnect(RESET1 := TRUE);
		RsStartConnect(RESET1 := FALSE);
	END_IF
END_IF

Out_Connected := SQLDatabase.bConnected;
END_METHOD

END_FUNCTION_BLOCK

// ---- 00_FunctionsBlocks/Database/Firebird/Firebird_WriteAlarms.TcPOU
PROGRAM Firebird_WriteAlarms
VAR_INPUT
	ParamTimeBetweenReconnect	: TIME := T#1M;
	IN_Reset					: BOOL;
	
	FIFO						: FB_DBDatasetFifo;
END_VAR
VAR_OUTPUT
END_VAR
	
VAR

	CmdStart					: BOOL;
	CmdReset					: BOOL;
	// Data processing 
	MesDataExd			: LoggerFirebird ; 
	// RESET
		Trig_Reset				: R_TRIG;
		
	// Connexion
		TP_Reconnect			: TP;
		Trig_Connect			: R_TRIG;
		RS_Connect				: RS;
		RS_HasBeenConnected		: RS;
	// DISCONNECT
		TrigStartDisconnect				: R_TRIG;
		RsStartDisconnect				: RS;		
		
		
	// Write File       
		ETAPE					: UINT;
		Trig_Start				: R_TRIG;   
		Requete					: STRING(1000);
		sTimeStamp 				: STRING(255);
		sTimeStamp_Ms			: STRING(255);
		sValue					: STRING(255);
		sAck					: STRING(255);
		Format					: FB_FormatString;
		SQLDatabase				: FB_SQLDatabaseEvt('',T#10S);
		SQLCommand1				: FB_SQLCommandEvt('',T#10S);
		SQLCommandNull			: FB_SQLCommandEvt('',T#10S);
		
	
	// General variables
		bInit 					: BOOL;

		NomTable				: STRING(255) := 'TABLE_ALARMS';
		

	
END_VAR

// DataProcessing
IF NOT bInit THEN
	M_Init();
END_IF
RS_HasBeenConnected(SET := SQLDatabase.bConnected);
TP_Reconnect(In :=RS_HasBeenConnected.Q1 AND NOT SQLDatabase.bConnected OR NOT bInit OR TP_Reconnect.Q, PT := ParamTimeBetweenReconnect);
	
M_AlarmManager();


Trig_Reset(CLK := IN_Reset OR CmdClearFault_G);
IF Trig_Reset.Q THEN
	FIFO.A_Reset();
	SQLCommand1 := SQLCommandNull;
	CmdReset := False;
END_IF


// La première ligne est non nulle
CmdStart := FIFO.nCount >0 AND SQLDatabase.bConnected;
Trig_Start(CLK := CmdStart);
IF Trig_Start.Q THEN
	ETAPE := 1;
END_IF
		
CASE ETAPE OF
	1: // CONNECTED
		IF SQLDatabase.CreateCmd(pSQLCommand := ADR(SQLCommand1)) THEN 
			IF NOT SQLCommand1.bError THEN
				ETAPE := 2;
			ELSIF SQLCommand1.bError THEN
				ETAPE := 255;
			END_IF
		END_IF
		
	2:
		//sTimeStamp := left(STR := (AX_Buffer_Alarms[1].TimeStamp_Act), SIZE := LEN((AX_Buffer_Alarms[1].TimeStamp_Act))-4);
		FIFO.A_Get();	
		sTimeStamp := FIFO.OUT.TimeStamp_Act;
		sTimeStamp_MS := right(STR := (sTimeStamp), SIZE := 3);	
		sValue	:= INT_TO_STRING(BOOL_TO_INT(FIFO.Out.Value));
		sAck	:= INT_TO_STRING(BOOL_TO_INT(FIFO.Out.Ack));
		Format(sFormat := 'Insert into %s values ( $'%s$',%d, %s, %s);', 
			sOut => Requete,
			arg1 := F_STRING(in := NomTable),
			arg2 := F_STRING(in := sTimeStamp),
			arg3 := F_UINT(in := FIFO.Out.ID),
			arg4 := F_STRING(in := sValue),
			arg5 := F_STRING(in := sAck)
		);
		IF SQLCommand1.Execute(pSQLCmd := ADR(Requete), cbSQLCmd := SIZEOF(Requete))THEN
			IF  NOT SQLCommand1.bError THEN
				ETAPE := 4;
			ELSIF SQLCommand1.bError THEN
				ETAPE := 255;
			END_IF
		END_IF

	4:
		IF NOT SQLDatabase.bError THEN
			FIFO.A_Remove();
			Requete  := '';
			Trig_Start(CLK := FALSE);
			Etape := 0;
		ELSE 
			ETAPE := 255;
		END_IF
		
	255: 
		CmdReset := TRUE;
		Requete := '';
		Etape := 0;
		CmdStart := FALSE;
END_CASE

METHOD M_AlarmManager
VAR
	FB_AlarmCodeManager : FB_AlarmCodeManager;
END_VAR
// Gestion des alarmes internes au code

FB_AlarmCodeManager
(
	bAlarm1 := SQLCommand1.bError,				// Insert new alarm failed
	bAlarm2 := SQLDatabase.bError,				// Connexion to database failed
	bAlarm3 := FALSE,							// 
	bAlarm4 := FIFO.bOverwrite,					// Fifo Overflow
	bAlarm5 :=FALSE,							//
	bAlarm6 :=FALSE,    						//
	bAlarm7 :=FALSE,    						//
	bAlarm8 :=FALSE,    						//
	bAlarm9 :=FALSE,    						//
	bAlarm10 :=FALSE,   						//
	bAlarm11 :=FALSE,   						//
	bAlarm12 :=FALSE,   						//
	bAlarm13 :=FALSE,   						//
	bAlarm14 :=FALSE,   						//
	bAlarm15 :=FALSE,							//	
	
	wAlarmCode =>MesDataExd.MesData.MesAlarmCode
);
END_METHOD

METHOD M_Connect : BOOL

VAR_OUTPUT
END_VAR
VAR_INPUT
	IN_hDBID				: DINT;
	IN_Start				: BOOL;
END_VAR
Trig_Connect(CLK := IN_Start);
RS_Connect(SET := Trig_Connect.Q);
IF RS_Connect.Q1 THEN
	IF SQLDatabase.Connect(hDBID := IN_hDBID) THEN;
		RS_Connect(RESET1 := TRUE);
		RS_Connect(RESET1 := FALSE);
	END_IF
END_IF
END_METHOD

METHOD M_Disconnect : BOOL
VAR_INPUT
END_VAR
VAR_INPUT
	IN_Start				: BOOL;
END_VAR
VAR
END_VAR
TrigStartDisconnect(CLK := IN_Start);
RsStartDisconnect(SET := TrigStartDisconnect.Q);
IF RsStartDisconnect.Q1 THEN
	IF SQLDatabase.Disconnect() THEN;
		RsStartDisconnect(RESET1 := TRUE);
		RsStartDisconnect(RESET1 := FALSE);
	END_IF
END_IF
END_METHOD

METHOD M_Init

VAR
	LL	: SINT;
	KK 	: SINT;
END_VAR
//Initialisation BUFFER
	//Buffer pour la lecture des sms
	FIFO.A_Reset();
	FIFO.A_Add();
	FIFO.A_Get();
	FIFO.A_Remove();
	
	FIFO.In.Message :=  'Activation du code';
	FIFO.In.TimeStamp_Act := SYSTEMTIME_TO_STRING(CalLocalTimeStruct); 
	FIFO.A_Add();
	bInit := TRUE;
END_METHOD

END_PROGRAM

// ---- 00_FunctionsBlocks/Database/InfluxDb/InfluxDb_AlarmsManagement.TcPOU
PROGRAM InfluxDb_AlarmsManagement

VAR_INPUT
	IN_FIFO										: FB_DBDatasetFifo;
	IN_Reset									: BOOL;
	//MesDataExd								: LoggerInfluxDb;
END_VAR

VAR
	// M_Init
   		bInit 									: BOOL;
	// Reset                					
		Trig_Reset								: R_TRIG;
	// Interface values
		bGet: BOOL;
		bRem: BOOL;
		Out_Alarms 				: ST_ValuesAlarms;
		Out_Alarms_Null 		: ST_ValuesAlarms;
END_VAR

IF NOT bInit THEN
	M_Init();
END_IF

Trig_Reset(CLK := IN_Reset OR CmdClearFault_G);
IF Trig_Reset.Q THEN
	IN_Reset := FALSE;
	IN_FIFO.A_Reset();
	Out_Alarms := Out_Alarms_Null;
END_IF

IF bRem THEN
	bRem := FALSE;
	IN_FIFO.A_Remove();
	Out_Alarms := Out_Alarms_Null;
END_IF

IF bGet THEN
	bGet := FALSE;
	IN_FIFO.A_Get();
	Out_Alarms := IN_FIFO.Out;
END_IF

METHOD M_Init : BOOL
VAR_INPUT
END_VAR
//Initialisation BUFFER
	//Buffer pour la lecture des sms
	//IN_FIFO.A_Reset();
	//IN_FIFO.A_Add();
	//IN_FIFO.A_Get();
	//IN_FIFO.A_Remove();
	
	IN_FIFO.In.Message :=  'Code Activation';
	IN_FIFO.IN.TimeStamp_Act := SYSTEMTIME_TO_STRING(CalLocalTimeStruct);
	IN_FIFO.A_Add();
	bInit := TRUE;
END_METHOD

END_PROGRAM

// ---- 00_FunctionsBlocks/Database/InfluxDb/InfluxDb_ReadValues.TcPOU
PROGRAM InfluxDb_ReadValues
               					
VAR_INPUT  
	IN_TimeStart							: LINT;
	IN_bRead								: BOOL;             					
	IN_Dbid									: UINT := 1;
	IN_NbRecordRead							: UINT := 100;
	IN_bAck									: BOOL;	// Filter value for acknowledged filter
	IN_bVal									: BOOL; // Filter value for value filter
	IN_FilterAck							: BOOL; // Is the acknowledged filter active 
	IN_FilterVal							: BOOL; // Is the value filter active 
	IN_Database								: T_MaxString;
END_VAR

VAR_OUTPUT
    OUT_bError								: BOOL;
	OUT_bBusy								: BOOL;
	OUT_pTableResults						: PVOID;
	OUT_cbTableResults						: UINT;
END_VAR

VAR
	Query									: T_MaxString;
	QueryInit								: T_MaxString := 'SELECT time, Message, ID, Value, Ack  FROM %s.autogen.Alarms  ';
	QueryOrder								: T_MaxString := ' order by time desc limit %d';
	QueryFinal								: T_MaxString ;
	
    QueryOption_TSDB_Select 				: T_QueryOptionTimeSeriesDB_Query; 
    fbNoSQLQueryBuilder_TimeSeriesDB 		: FB_NoSQLQueryBuilder_TimeSeriesDB; 
    fbNoSqlQueryEvt 						: FB_NoSQLQueryEvt(sNetID := '', tTimeout := T#15S); 
	fbNoSqlResultEvt						: FB_NoSQLResultEvt(sNetID := '', tTimeout := T#15S);
	fbNoSqlValidationEvt					: FB_NoSQLValidationEvt(sNetID := '', tTimeout := T#15S);
	nState 									: UINT;
	ReaDS_Transfouct								: ARRAY[1..250]OF ST_InfluxAlarmsRetrieve;
	Format									: FB_FormatString;          						

END_VAR

fbNoSQLQueryBuilder_TimeSeriesDB.pQueryOptions := ADR(QueryOption_TSDB_Select);
fbNoSQLQueryBuilder_TimeSeriesDB.cbQueryOptions := SIZEOF(QueryOption_TSDB_Select);

OUT_pTableResults 	:= ADR(ReaDS_Transfouct);
OUT_cbTableResults 	:= SIZEOF(ReaDS_Transfouct);

IF IN_bRead THEN
	OUT_bBusy 	:= TRUE;
	IN_bRead 	:= FALSE;
	nState 		:= 1;
	Query := QueryInit;
	IF IN_FilterAck OR IN_FilterVal THEN
		query := concat(STR1 := query, str2 := 'Where ');
		
		IF IN_FilterAck THEN
			query := concat(STR1:= query, STR2 := concat(STR1 := ' Ack=', str2 := BOOL_TO_STRING(IN_bAck)));
		END_IF
		
		IF IN_FilterAck AND IN_FilterVal THEN
			query := concat(STR1:= query, STR2 := ' AND ');
		END_IF
		
		IF IN_FilterVal THEN
			query := concat(STR1:= query, STR2 := concat(STR1 := 'Value=', str2 := BOOL_TO_STRING(IN_bVal)));
		END_IF
		
	END_IF
	query := concat(str1 := query, STR2 := QueryOrder);
	Format(sFormat := Query, arg1 := F_STRING(in:=IN_Database), arg2:= F_UINT(in:=IN_NbRecordRead), sOut => QueryFinal);
	
	QueryOption_TSDB_Select.cbQuery := SIZEOF(QueryFinal);
	QueryOption_TSDB_Select.pQuery := ADR(QueryFinal);
END_IF

CASE nState OF 
	1:
		IF fbNoSqlQueryEvt.ExecuteDataReturn(hDBID := IN_Dbid, iNoSQLQueryBuilder := fbNoSQLQueryBuilder_TimeSeriesDB, pNoSQLResult := ADR(fbNoSqlResultEvt)) THEN
			IF fbNoSqlQueryEvt.bError THEN
				OUT_bError := TRUE;
				nState := 0;
			ELSE
				nState := 2;
			END_IF
		END_IF
	2:
		IF fbNoSqlResultEvt.ReadAsStruct
		(
			nStartIndex := 0, 
			nRecordCount:= IN_NbRecordRead,  
			pData:= ADR(ReaDS_Transfouct),  
			cbData:= SIZEOF(ReaDS_Transfouct),  
			bValidate := TRUE,  
			bDataRelease:= TRUE,  
			pNoSQLValidation:= ADR(fbNoSqlValidationEvt) 
		) THEN
			IF fbNoSqlResultEvt.bError THEN
				OUT_bError := TRUE;
				OUT_bBusy := FALSE;
				nState := 0;
			ELSE
				nState := 3;
				OUT_bBusy := FALSE;
			END_IF
		END_IF
	
END_CASE

END_PROGRAM

// ---- 00_FunctionsBlocks/Database/InfluxDb/InfluxDb_WriteAlarms.TcPOU
PROGRAM InfluxDb_WriteAlarms

VAR_INPUT
	IN_Dbid										: UINT;
	IN_FIFO										: FB_DBDatasetFifo_Influx;
	IN_Reset									: BOOL;
MesDataExd								: LoggerInfluxDb;
END_VAR

VAR
	// M_Init
		TP_Init									: TP;
		F_TRIG_Init								: F_TRIG;
   		bInit 									: BOOL;
	// Reset                					
		Trig_Reset								: R_TRIG;
	// Insert value             				
		CmdStart								: BOOL;
    	QueryOption_TSDB_Insert 				: T_QueryOptionTimeSeriesDB_Insert; // defines detailed Queryparameter
    	fbNoSQLQueryBuilder_TimeSeriesDB 		: FB_NoSQLQueryBuilder_TimeSeriesDB; // defines database type specific api
    	fbNoSqlQueryEvt 						: FB_NoSQLQueryEvt(sNetID := '', tTimeout := T#15S); // functionblock to execute queries
		nState 									: UINT;
		ValueToInsert							: ST_InfluxAlarmsInsert;
    // error handling helper values
    sErrorMessage								: STRING(255);

	
END_VAR

IF NOT bInit THEN
	M_Init();
END_IF

Trig_Reset(CLK := IN_Reset OR CmdClearFault_G);
IF Trig_Reset.Q THEN
	IN_Reset := FALSE;
	IN_FIFO.A_Reset();
END_IF

CmdStart := IN_FIFO.nCount >0 ;
IF CmdStart THEN
	CmdStart := FALSE;
	
	fbNoSQLQueryBuilder_TimeSeriesDB.pQueryOptions := ADR(QueryOption_TSDB_Insert);
	fbNoSQLQueryBuilder_TimeSeriesDB.cbQueryOptions := SIZEOF(QueryOption_TSDB_Insert);
	IN_FIFO.A_Get();
	ValueToInsert	:= IN_FIFO.Out;
	QueryOption_TSDB_Insert.sTableName 			:= 'Alarms';			
	QueryOption_TSDB_Insert.sDataType 			:= 'ST_InfluxAlarmsInsert';	
	QueryOption_TSDB_Insert.pSymbol 			:= ADR(ValueToInsert); 	
	QueryOption_TSDB_Insert.cbSymbol 			:= SIZEOF(ValueToInsert); 
	QueryOption_TSDB_Insert.nDataCount 			:= 1;					
	QueryOption_TSDB_Insert.nStartTimestamp 	:= F_GetSystemTime(); 	

	nState := 3;
END_IF

CASE nState OF 
    3:
        IF fbNoSqlQueryEvt.Execute(IN_Dbid, fbNoSQLQueryBuilder_TimeSeriesDB) THEN
			IF fbNoSqlQueryEvt.bError THEN
			MesDataExd.MesData.MesAlarmCode.1 := TRUE;
				nState := 1;
			ELSE
			MesDataExd.MesData.MesAlarmCode.1 := FALSE;
			   	nState := 1;
 				IN_FIFO.A_Remove();
           END_IF
        END_IF
END_CASE

METHOD M_Init : BOOL
VAR_INPUT
END_VAR
//Initialisation BUFFER
	//Buffer pour la lecture des sms
	IN_FIFO.A_Reset();
	IN_FIFO.A_Add();
	IN_FIFO.A_Get();
	IN_FIFO.A_Remove();
	
	IN_FIFO.In.Message :=  'Activation du code';
	IN_FIFO.A_Add();
	bInit := TRUE;
END_METHOD

END_PROGRAM

// ---- 00_FunctionsBlocks/Database/InfluxDb/InfluxDb_WriteStruct.TcPOU
FUNCTION_BLOCK InfluxDb_WriteStruct
VAR_INPUT PERSISTENT
	ParamInitTime							: TIME := T#1S;
END_VAR                 					
VAR_INPUT               					
	IN_Table 								: STRING;
	IN_StructureName 						: STRING;
	IN_DataAddr								: PVOID;
	IN_DataSize								: UDINT;
	IN_NumberStructure						: UDINT;		// ArrayLength
	IN_DataFrequency						: TIME;
	IN_Dbid									: UINT;
END_VAR

VAR
    QueryOption_TSDB_Insert 				: T_QueryOptionTimeSeriesDB_Insert; // defines detailed Queryparameter
    fbNoSQLQueryBuilder_TimeSeriesDB 		: FB_NoSQLQueryBuilder_TimeSeriesDB; // defines database type specific api
    fbNoSqlQueryEvt 						: FB_NoSQLQueryEvt(sNetID := '', tTimeout := T#15S); // functionblock to execute queries
    bInit 									: BOOL;
	nState 									: UINT;
    Name 									: STRING;
	Current_Time 							: TIME;
	Old_Time	 							: TIME;
	
    // error handling helper values
    bError									: BOOL;
    sErrorMessage							: STRING(255);
                    						
	// InitWait     						
	TP_Init									: TP;
	F_TRIG_Init								: F_TRIG;
	
END_VAR

fbNoSQLQueryBuilder_TimeSeriesDB.pQueryOptions := ADR(QueryOption_TSDB_Insert);
fbNoSQLQueryBuilder_TimeSeriesDB.cbQueryOptions := SIZEOF(QueryOption_TSDB_Insert);

QueryOption_TSDB_Insert.sTableName 			:= IN_Table;			//'PcsTable1';
QueryOption_TSDB_Insert.sDataType 			:= IN_StructureName;	//'ST_Pcs';
QueryOption_TSDB_Insert.pSymbol 			:= IN_DataAddr; 		//ADR(AX_InvData);
QueryOption_TSDB_Insert.cbSymbol 			:= IN_DataSize; 		//SIZEOF(AX_InvData);
QueryOption_TSDB_Insert.nDataCount 			:= IN_NumberStructure;	//CstNbInv*CstNbPcs_Inv; 
QueryOption_TSDB_Insert.nStartTimestamp 	:= F_GetSystemTime(); 	// get current twincat time 
QueryOption_TSDB_Insert.nCycleTime		 	:= 0; 					// 0 : insert all structures at the same time

TP_Init(IN := NOT bInit OR CmdInit_G, PT := ParamInitTime);
F_TRIG_Init(CLK := TP_Init.Q);
IF F_TRIG_Init.Q THEN
	nState := 1;
END_IF


CASE nState OF 
    1: // init 
		Current_Time := TIME();
		IF Current_Time > Old_Time + IN_DataFrequency - INT_TO_TIME(CstCycleTime_G) THEN
			nState := 3;
			
		END_IF
    3: // write values 
		Old_Time := TIME();
        IF fbNoSqlQueryEvt.Execute(IN_Dbid, fbNoSQLQueryBuilder_TimeSeriesDB) THEN
            IF fbNoSqlQueryEvt.bError THEN
               bError := TRUE;
			   nState := 1;
            ELSE
				bError := FALSE;
			   	nState := 1;
            END_IF
        END_IF
	
END_CASE

END_FUNCTION_BLOCK

// ---- 00_FunctionsBlocks/Database/PRG_EpochConverter.TcPOU
PROGRAM PRG_EpochConverter
//Convert Epoch to TimeStruct
VAR
	FileTime				: T_FILETIME;
	ConvertTime				: FB_SystemTimeToTzSpecificLocalTime;
END_VAR
VAR_INPUT
	IN_bIsWeird 			: BOOL; 				// Cas pour l'Epoch venant de Influx : offset de   82 011 087 
	IN_OffSet				: DINT :=  -82011087 ; 	// Cas pour l'Epoch venant de Influx : valeur de l'offset
	IN_Epoch				: LINT;					// Input 
END_VAR             		
VAR_OUTPUT          		
	OUT_TimeStruct_UTC		: TIMESTRUCT;
	OUT_TimeStruct_Local	: TIMESTRUCT;
END_VAR

IF IN_bIsWeird THEN
	IN_Epoch := IN_Epoch + IN_OffSet;
END_IF

FileTime.dwHighDateTime := LINT_TO_DWORD(SHR(IN_Epoch, 32));
FileTime.dwLowDateTime 	:= LINT_TO_DWORD(IN_Epoch);
OUT_TimeStruct_UTC 		:= FILETIME_TO_SYSTEMTIME( FileTime );
ConvertTime(in := OUT_TimeStruct_UTC, tzInfo := CstTimeZone_G, out => OUT_TimeStruct_Local);

END_PROGRAM

// ---- 00_FunctionsBlocks/Database/PRG_TimestructConverter.TcPOU
PROGRAM PRG_TimestructConverter
//Convert TimeStruct to Epoch 
VAR
	DT_Time			: DT;
	FileTime		: T_FILETIME;
END_VAR
VAR_INPUT
	IN_TimeStruct			: TIMESTRUCT;					// Input 
END_VAR             		
VAR_OUTPUT          		
	OUT_Epoch		: LINT;
END_VAR

DT_Time 		:= SYSTEMTIME_TO_DT( IN_TimeStruct );

FileTime 		:= DT_TO_FILETIME(dtIn := DT_Time);

OUT_Epoch := (SHL(DWORD_TO_ULINT(FileTime.dwHighDateTime), 32) + DWORD_TO_ULINT(FileTime.dwLowDateTime)) / 10000000 - 11644473600;

END_PROGRAM

// ---- 00_FunctionsBlocks/Database/SQLCe/FB_SQLExpert_InsertBuffer_1.TcPOU
FUNCTION_BLOCK FB_SQLExpert_InsertBuffer_1
// Fonctionnement : Tableau de 2000 structures en input. Dès qu'on atteint 1000 structures remplies, décalage de l'espace mémoire
// pour en 1 temps de cycle pour ne pas perdre de données sur le transfert.
VAR CONSTANT
	CstNbLigneBuffer		: DINT:= 500;
	CstNbLigneBufferMax	 	: DINT:= 5000;

END_VAR

VAR_INPUT
	NomTable				: STRING := 'Table100ms';
	hDBID					: UDINT;
END_VAR

